// TwinCAT 3 PLC project PLC
// ProgramVersion: 3.1.4026.9
// CompilerDefines: {define InputField}{define ThirdOutputField}
// libraries:
//   Tc2_ControllerToolbox, * (Beckhoff Automation GmbH)
//   Tc2_ModbusRTU, * (Beckhoff Automation GmbH)
//   Tc2_ModbusSrv, * (Beckhoff Automation GmbH)
//   Tc2_Standard, * (Beckhoff Automation GmbH)
//   Tc2_System, * (Beckhoff Automation GmbH)
//   Tc2_Utilities, * (Beckhoff Automation GmbH)
//   Tc3_Module, * (Beckhoff Automation GmbH)
// project tree:
//   GVLs/ Config.TcGVL, GVL.TcGVL
//   / PlcTask.TcTTO
//   POUs/ErrorHandling/ eErrAckAccess.TcDUT, ErrorHandling.TcPOU, eSeverity.TcDUT, FB_AddErrorST.TcPOU, ST_ErrorStruct.TcDUT
//   POUs/ErrorHandling/New eventlogger %28TBD%29/ EventLogger.TcPOU (not stored), FB_Alarm.TcPOU (not stored), fb_EventAlarm.TcPOU (not stored)
//   POUs/FunctionBlocks/ fbDwordToReal.TcPOU, fbRealToDWord.TcPOU, fbRealToWord.TcPOU, fbWordToReal.TcPOU
//   POUs/ MAIN.TcPOU, POU.TcPOU
//   POUs/MonitoringControl/ FB_ControlManager.TcPOU
//   POUs/MonitoringControl/ProfinetController/enums/ e_controllerStatus.TcDUT
//   POUs/MonitoringControl/ProfinetController/ FB_PNController.TcPOU (excluded from build)
//   POUs/MonitoringControl/ProfinetController/Structs/future use/ ST_PNInput_DCBusExpansion.TcDUT, ST_PNInput_DCCharger.TcDUT, ST_PNInput_ParallelOperation.TcDUT, ST_PNOutput_DCCharger.TcDUT, ST_PNOutput_DCExpansion.TcDUT, ST_PNOutput_ParallelOperation.TcDUT
//   POUs/MonitoringControl/ProfinetController/Structs/ STParams.TcDUT, ST_PNController_Events.TcDUT, ST_PNController_Get.TcDUT, ST_PNController_Set.TcDUT, ST_PNInput_Battery.TcDUT, ST_PNInput_General.TcDUT, ST_PNInput_InputField.TcDUT, ST_PNInput_PeakShaveBox.TcDUT, ST_PNInput_Powerstack.TcDUT, ST_PNOutput_Battery.TcDUT, ST_PNOutput_General.TcDUT, ST_PNOutput_InputField.TcDUT, ST_PNOutput_OutputField.TcDUT, ST_PNOutput_PeakShaveBox.TcDUT, ST_PNOutput_PowerStack.TcDUT, ST_PNOutput_ZPT.TcDUT
//   POUs/Objects/BMS/eNums/ eBMS_Status.TcDUT, eHVDC_Powerstatus.TcDUT, ePOUState.TcDUT, ePowerControl.TcDUT, ePowerOnStatus.TcDUT, eSubValues.TcDUT
//   POUs/Objects/BMS/ FB_BMS.TcPOU, FB_BMS_IO.TcPOU
//   POUs/Objects/BMS/Structs/ st_BMS_Events.TcDUT, st_BMS_GetStatus.TcDUT, st_BMS_IO.TcDUT, st_BMS_Set.TcDUT, st_MBMU_BatterySummary.TcDUT, st_MBMU_Status.TcDUT, st_SBMU_BatterySummary.TcDUT, st_SBMU_Status.TcDUT
//   POUs/Objects/CoolingSystem/CoolingStack/eNums/ eHeatPumpMode.TcDUT, eHeatPumpState.TcDUT
//   POUs/Objects/CoolingSystem/CoolingStack/ FB_Heatpump.TcPOU, FB_HeatPumpSystem.TcPOU, FB_Heatpumpsystem_IO.TcPOU
//   POUs/Objects/CoolingSystem/CoolingStack/SFC/ FB_HeatpumpInit.TcPOU, FB_HeatpumpOperation.TcPOU
//   POUs/Objects/CoolingSystem/CoolingStack/Structs/ ST_HeatPumpSystemEvents.TcDUT, ST_HeatpumpSystemGet.TcDUT, ST_HeatpumpData.TcDUT, ST_HeatPumpEvents.TcDUT, ST_HeatPumpGet.TcDUT, st_OperatingPoint.TcDUT
//   POUs/Objects/CoolingSystem/ CoolingSystemParams.TcGVL, FB_CoolingSystem.TcPOU, FB_CoolingSystem_IO.TcPOU
//   POUs/Objects/CoolingSystem/SFC/Enums/ eConditioningRequirement.TcDUT, eConditioningStates.TcDUT
//   POUs/Objects/CoolingSystem/SFC/ FB_BatteryConditioningSFC.TcPOU, FB_DehumidifySFC.TcPOU, FB_EnclosureConditioningSFC.TcPOU, FB_PowerModeConditioningSFC.TcPOU
//   POUs/Objects/CoolingSystem/Structs/ ST_ConditioningRequirements.TcDUT, ST_CoolingSystemEvents.TcDUT, ST_CoolingSystemGet.TcDUT, ST_CoolingSystemInputs.TcDUT, ST_CoolingSystemOutputs.TcDUT, ST_CoolingSystem_Control.TcDUT, ST_SensorValues.TcDUT
//   POUs/Objects/ExternalControl/ FB_ExternalControl.TcPOU
//   POUs/Objects/InternalPowerSupply/eNums/ ePowerStatus.TcDUT, eSupplyState.TcDUT
//   POUs/Objects/InternalPowerSupply/ FB_InternalPowerSupply.TcPOU, FB_InternalPowerSupply_IO.TcPOU, IPSParams.TcGVL
//   POUs/Objects/InternalPowerSupply/Structs/ ST_InternalPowerStatus.TcDUT, ST_InternalPowerSupply_Events.TcDUT, ST_InternalPowerSupply_Get.TcDUT, ST_InternalPowersupply_set.TcDUT, ST_PowerDemand.TcDUT
//   POUs/Objects/InternalPowerSupply/UPS/eNums/ eUPSState.TcDUT
//   POUs/Objects/InternalPowerSupply/UPS/ FB_UPS.TcPOU
//   POUs/Objects/InternalPowerSupply/UPS/Structs/ ST_UPSData.TcDUT, ST_UPSEvents.TcDUT, ST_UPSGET.TcDUT
//   POUs/Objects/LedstripController/ eLedStripCommands.TcDUT, UpdateSFC.TcPOU
//   POUs/Objects/LedstripController/Structs/ stLedControl.TcDUT, stLedStatus.TcDUT, st_LedColor.TcDUT, ST_Ledstrip_IOvars.TcDUT, u_LedColor.TcDUT
//   POUs/Objects/PowerQualityMonitor/FB_Beckhoff_EL3443_0010/ FB_EL3443_0010.TcPOU, ST_EL3443_PhaseStatus.TcDUT, ST_EL3443_TotalStatus.TcDUT
//   POUs/Objects/PowerQualityMonitor/FB_Janitza_UMG801/ FB_Janitza.TcPOU, PowerMeterConfig.TcGVL, ST_Powerlockdata.TcDUT
//   POUs/Objects/PowerQualityMonitor/ FB_PowerQualityMonitoring.TcPOU
//   POUs/Objects/PowerQualityMonitor/_Enums/ eACRotationState.TcDUT, Phases.TcDUT
//   POUs/Objects/PowerQualityMonitor/_Structs/ ST_InputVoltageMeter.TcDUT, ST_PowerMonitor_BESS.TcDUT, ST_PowerMonitor_Events.TcDUT, ST_PowerMonitor_get.TcDUT, ST_PowerMonitor_InputField.TcDUT, ST_PowerMonitor_Internal.TcDUT, ST_PowerMonitor_OutputField.TcDUT
//   POUs/Objects/PowerStack/eNums/ eNetcontactorState.TcDUT, eStatus.TcDUT
//   POUs/Objects/PowerStack/ st_Powerstack_get.TcDUT
//   POUs/Objects/ProtectionSystems/FireDetection/eNums/ eFireAlarmStatus.TcDUT, eCOAlarmStatus.TcDUT
//   POUs/Objects/ProtectionSystems/FireDetection/ FB_FireDetection.TcPOU, FB_FireDetection_IO.TcPOU
//   POUs/Objects/ProtectionSystems/FireDetection/Structs/ ST_COInputData.TcDUT, ST_FireDetectionGet.TcDUT, ST_FireDetectionSet.TcDUT, ST_FireSystem_Events.TcDUT, ST_SmokeDetIO.TcDUT
//   POUs/Objects/RouterData/ FB_Teltonika.TcPOU
//   POUs/Objects/RouterData/Struct/ dwtoreal.TcDUT, eSMSStatus.TcDUT, st_Device.TcDUT, st_GPS.TcDUT, st_mobile.TcDUT, st_router_data.TcDUT, ST_Router_params.TcDUT, st_TeltonikaEvents.TcDUT
//   POUs/old/ old.TcPOU
//   POUs/ProfinetHandling/ InitSIEMENSInput.TcPOU, SetSiemensControlModes.TcPOU, SetSIEMENSOutput.TcPOU, SiemensControl.TcPOU
//   POUs/System/_Structs/ ST_SystemControl_FromSystem.TcDUT
//   POUs/System/_Structs/TempStructs/ eCOAlarmStatus_1.TcDUT, eSmokeDetectAlarmStatus.TcDUT, eWago750495_ACDataID.TcDUT, eWago750495_HarmonicsDataID.TcDUT, eWago750495_MeasureGroupID.TcDUT, eWago750495_StatDataID.TcDUT, ST_ACSwitchgear_Get.TcDUT, ST_CODetectors.TcDUT, ST_DCSwitchgear_Get.TcDUT, ST_Enclosure_get.TcDUT, ST_FireDetection_get.TcDUT, ST_FireDetection_get_1.TcDUT, ST_FireDetection_set.TcDUT, ST_FireSystem_Events_1.TcDUT, ST_FireSystem_Events_2.TcDUT, ST_InsulationMonitor_get.TcDUT, ST_NeutralTransformer_Get.TcDUT, ST_OvercurrentProtection_get.TcDUT, ST_PeakShaveBox_Get.TcDUT, ST_PLCstate_get.TcDUT, ST_ProtectionSystems_get.TcDUT, ST_ResidualCurrentMonitor_get.TcDUT, ST_Safety_get.TcDUT, ST_Safety_get_1.TcDUT, ST_SmokeDetectors.TcDUT, ST_SmokeDetIO_1.TcDUT, ST_Surgeprotection_get.TcDUT, ST_SystemControl_System.TcDUT, ST_System_Properties.TcDUT, ST_Wago750354_get.TcDUT, ST_Wago750495_Data.TcDUT, ST_Wago750495_ExtStatusWord.TcDUT, ST_Wago750495_Get.TcDUT, ST_Wago750495_Set.TcDUT, ST_Wago750495_StatusWord.TcDUT
// real-time tasks:
//   TASK PlcTask: cycle T#4ms, priority 1, ADS port 350
// I/O:
//   DEVICE Device 1 (EtherCAT), AmsNetId 5.131.105.63.2.1
//     Term 2 (EK1200) [EK1200-5000 EtherCAT Power supply (2A E-Bus)]
//       Term 2 (EL6070-0033) [EL6070-0033 1Ch. Licence key terminal, individual licences]
//       Term 25 (EL2574) [EL2574 4 Ch. Pixel LED Controller]
//         modules: SlotGroup 1 (Slot 1, 2), SlotGroup 1 (Slot 1, 2), SlotGroup 2 (Slot 3, 4), SlotGroup 2 (Slot 3, 4)
//       Term 3 (EL1809) [EL1809 16Ch. Dig. Input 24V, 3ms]
//       Term 4 (EL1809) [EL1809 16Ch. Dig. Input 24V, 3ms]
//       Term 6 (EL2809) [EL2809 16Ch. Dig. Output 24V, 0.5A]
//       Term 8 (EL2809) [EL2809 16Ch. Dig. Output 24V, 0.5A]
//       Term 9 (EL3054) [EL3054 4Ch. Ana. Input 4-20mA]
//       Term 10 (EL3054) [EL3054 4Ch. Ana. Input 4-20mA]
//       Term 11 (EL6021) [EL6021 Schnittstelle (RS422/485)]
//       Term 12 (EL3443-0010) [EL3443-0010 3Ch. Power Measuring 10A]
//       Term 13 (EL4002) [EL4002 2K. Ana. Ausgang 0-10V, 12bit]
//       Term 14 (EL1918) [EL1918, 8Ch. Safety Input 24V, TwinSAFE]
//         modules: Module 1 (FSOE), Module 2 (FSLOGIC)
//       Term 15 (EL2904) [EL2904, 4 Ch. Safety Output 24V, 0.5A, TwinSAFE]
//         modules: Module 1 (FSOES), Module 2 (DO)
//       Term 16 (EK1122) [EK1122 2 port EtherCAT junction]
//       Term 16 (EL9011) [EL9011 End Terminal]
//   DEVICE Device 4 (USB) (disabled)
//   DEVICE Device 5 (COM Port) (disabled)
//   DEVICE Device 6 (NOV-DP-RAM)
//   DEVICE Device 2 (Profinet Controller), AmsNetId 5.131.105.63.3.1
//     pn-coupler [Helmholz GmbH & Co. KG PN/PN Coupler X1 (left network), firmware V2, 700-158-3PN02, supports Conformance Class A,B 700-158-3PN02] (disabled)
//       modules: Term 3 (DAP Module), Term 4 (IN  32 Bytes), Term 5 (IN  32 Bytes), Term 7 (IN  32 Bytes), Term 8 (IN  32 Bytes), Term 9 (IN  32 Bytes), Term 10 (IN  64 Bytes), Term 11 (IN  64 Bytes), Term 16 (OUT  32 Bytes), Term 15 (OUT  64 Bytes), Term 14 (OUT  64 Bytes), Term 13 (OUT  64 Bytes), InOutPowerData (OUT 128 Bytes)
//     quint4-ups-24dc-24dc-40-pn [Phoenix Contact PROFINET IO - Uninterruptible Power Supply 2907079] (disabled)
//       modules: Term 1 (DAP Module), Term 2 (QUINT4-UPS 24DC/40)
//     pnpncouplerx1 [Helmholz GmbH & Co. KG PN/PN Coupler X1 (left network), firmware V2, 700-158-3PN02, supports Conformance Class A,B 700-158-3PN02] (disabled)
//       modules: Term 17 (DAP Module), Term 18 (PeakShaveBox)
//     pnmbcold [Helmholz GmbH & Co. KG PN/ModbusTCP Coupler V2, supports Conformance Class A,B 700-159-3MB02] (disabled)
//       modules: Term 6 (DAP Module), Term 19 (Write Holding Register), Term 20 (Read Holding Register)
//     pnpncouplerx1-20 [Helmholz GmbH & Co. KG PN/PN Coupler X1 (left network), firmware V2, 700-158-3PN02, supports Conformance Class A,B 700-158-3PN02] (disabled)
//       modules: Term 21 (DAP Module), Term 22 (General), Term 23 (Battery), Term 24 (OutputField), Term 25 (InputField)
//     pninternal [VDL energy systems PN/PN Coupler X1 (left network), firmware V2, 700-158-3PN02, supports Conformance Class A,B PNController] (disabled)
//       modules: Term 26 (DAP Module), Term 28 (General), Term 29 (Battery), Term 30 (OutputField), Term 31 (InputGeneratorField), Term 32 (PowerstackField), Term 33 (PeakShaveBoxField), Term 34 (NeutralTransformerField)
//     pnexternal [VDL energy systems PN/PN Coupler X2 (right network), firmware V2, 700-158-3PN02, supports Conformance Class A,B PNController] (disabled)
//       modules: Term 27 (DAP Module), Term 35 (General), Term 36 (Battery), Term 37 (OutputField), Term 38 (InputGeneratorField), Term 39 (PowerstackField), Term 40 (NeutralTransformerField)
//     pnmbc2 [Helmholz GmbH & Co. KG PN/ModbusTCP Coupler V2, supports Conformance Class A,B 700-159-3MB02] (disabled)
//       modules: Term 41 (DAP Module), General.SystemState, General.Status, General.Warnings, General.Errors, General.CS_Status, General.CS_Warnings, General.CS_Errors, General.IPS_Status, General.IPS_Warnings, General.IPS_Errors, General.HeartbeatOut, General.Control, General.HeartbeatIn
//     pnmbc [Helmholz GmbH & Co. KG PN/ModbusTCP Coupler V2, supports Conformance Class A,B 700-159-3MB02]
//       modules: Term 41 (DAP Module), General_out, General_in, BMS_out, BMS_in, OutputField_out, InputField_out, InputField_in, PowerStack_out, PowerStack_in, PSB_out, PSB_in, ZPT_out
// variable links:
//   PLC/PLC Instance <-> Device 1 (EtherCAT)/Term 2 (EK1200)/Term 25 (EL2574)
//     PlcTask Inputs/MAIN.LedStripSFC.st_Status/b_CMDReject <-> SlotGroup 1 (Slot 1, 2)/Status Channel %C/Status/Command Reject
//     PlcTask Inputs/MAIN.LedStripSFC.st_Status/b_Error <-> SlotGroup 1 (Slot 1, 2)/Status Channel %C/Status/Error
//     PlcTask Inputs/MAIN.LedStripSFC.st_Status/b_SendAck <-> SlotGroup 1 (Slot 1, 2)/Status Channel %C/Status/Send Acknowledge
//     PlcTask Inputs/MAIN.LedStripSFC.st_Status/b_Transmit <-> SlotGroup 1 (Slot 1, 2)/Status Channel %C/Status/Transmit
//     PlcTask Inputs/MAIN.LedStripSFC.st_Status/b_UpdateAck <-> SlotGroup 1 (Slot 1, 2)/Status Channel %C/Status/Update Acknowledge
//     PlcTask Inputs/MAIN.LedStripSFC.st_Status/b_Warning <-> SlotGroup 1 (Slot 1, 2)/Status Channel %C/Status/Warning
//     PlcTask Inputs/MAIN.LedStripSFC.st_Status/b_busy <-> SlotGroup 1 (Slot 1, 2)/Status Channel %C/Status/Busy
//     PlcTask Outputs/MAIN.LedStripSFC.st_Control/b_Execute <-> SlotGroup 1 (Slot 1, 2)/Control Channel %C/Control/Execute
//     PlcTask Outputs/MAIN.LedStripSFC.st_Control/b_Send <-> SlotGroup 1 (Slot 1, 2)/Control Channel %C/Control/Send
//     PlcTask Outputs/MAIN.LedStripSFC.st_Control/b_Update <-> SlotGroup 1 (Slot 1, 2)/Control Channel %C/Control/Update
//     PlcTask Outputs/MAIN.LedStripSFC.st_Control/by_Command <-> SlotGroup 1 (Slot 1, 2)/Control Channel %C/Control/Command
//     PlcTask Outputs/MAIN.LedStripSFC.st_Control/dw_Color <-> SlotGroup 1 (Slot 1, 2)/Control Channel %C/Control/Color
//     PlcTask Outputs/MAIN.LedStripSFC.st_Control/w_Index <-> SlotGroup 1 (Slot 1, 2)/Control Channel %C/Control/Index
//     PlcTask Outputs/MAIN.LedStripSFC.st_Control/w_Length <-> SlotGroup 1 (Slot 1, 2)/Control Channel %C/Control/Length
//     PlcTask Outputs/MAIN.LedStripSFC.st_Control/w_Parameter <-> SlotGroup 1 (Slot 1, 2)/Control Channel %C/Control/Parameter
//   PLC/PLC Instance <-> Device 2 (Profinet Controller)/pnmbc2
//     PlcTask Inputs/MAIN.MBTestin <-> API/General.HeartbeatIn/Subterm 78 (Read Holding Register)/Inputs/General.HeartbeatIn
//     PlcTask Outputs/MAIN.MBTestOut <-> API/General.HeartbeatOut/Subterm 76 (Write Holding Register)/Outputs/General.HeartbeatOut

CONFIGURATION PLC
    RESOURCE PLC ON TwinCAT3
        TASK PlcTask(INTERVAL := T#4ms, PRIORITY := 1);
        PROGRAM MAIN WITH PlcTask : MAIN;
    END_RESOURCE
END_CONFIGURATION

// ---- POUs/ErrorHandling/eErrAckAccess.TcDUT
{attribute 'qualified_only'}
{attribute 'strict'}
TYPE eErrAckAccess :
(
	General := 0,
	Operator := 1,
	VDL := 2
);
END_TYPE

// ---- POUs/ErrorHandling/eSeverity.TcDUT
{attribute 'qualified_only'}
{attribute 'to_string'}
TYPE eSeverity :
(
	EmergencyShutdown			:= 0, //ONLY CALL FROM SAFETY PROGRAM
	QuickShutdown				:= 1,			
	NormalShutdown				:= 2,
	Warning 					:= 3,
	Info						:= 4
);
END_TYPE

// ---- POUs/ErrorHandling/ST_ErrorStruct.TcDUT
TYPE ST_ErrorStruct :
STRUCT
	b_ErrorActive	:BOOL;
	s_Severity 		:STRING(20);
	s_ID			:STRING(4);
	s_Message		:STRING(100);
	s_DateError		:STRING(20);
	s_TimeError		:STRING(20);
	s_TimeCleared	:STRING(20);
END_STRUCT
END_TYPE

// ---- POUs/MonitoringControl/ProfinetController/enums/e_controllerStatus.TcDUT
{attribute 'qualified_only'}
{attribute 'strict'}
TYPE e_controllerStatus :
(
	None 	:= 	0,
	Init	:=	1,
	Ready	:=	2,
	Active	:=	3,
	Error	:=	4
);
END_TYPE

// ---- POUs/MonitoringControl/ProfinetController/Structs/future use/ST_PNInput_DCBusExpansion.TcDUT
TYPE ST_PNInput_DCBusExpansion :
STRUCT
	ControlBits	:	DWORD;
END_STRUCT
END_TYPE

// ---- POUs/MonitoringControl/ProfinetController/Structs/future use/ST_PNInput_DCCharger.TcDUT
TYPE ST_PNInput_DCCharger :
STRUCT
	Controlbits	:	DWORD;
	//b_enable?
	//b_resetCharger
	//b_StartCharging
	Powerlimit	:	DWORD;
END_STRUCT
END_TYPE

// ---- POUs/MonitoringControl/ProfinetController/Structs/future use/ST_PNInput_ParallelOperation.TcDUT
TYPE ST_PNInput_ParallelOperation :
STRUCT
	Controlbits			:	DWORD;
	//b_DetectSlaves	
	r_ActivePower		:	DWORD;
	r_reactivePower		:	DWORD;
END_STRUCT
END_TYPE

// ---- POUs/MonitoringControl/ProfinetController/Structs/future use/ST_PNOutput_DCCharger.TcDUT
TYPE ST_PNOutput_DCCharger :
STRUCT
	statusbits		:	DWORD;
	ChargerStatus	:	DWORD;
	ChargePower		:	DWORD;
END_STRUCT
END_TYPE

// ---- POUs/MonitoringControl/ProfinetController/Structs/future use/ST_PNOutput_DCExpansion.TcDUT
TYPE ST_PNOutput_DCExpansion :
STRUCT
	statusbits	: DWORD;
	Busvoltage	: DWORD;
	RatedPower	: DWORD;
	LoadPercentage	: DWORD;
	CurrentPower	: DWORD;
END_STRUCT
END_TYPE

// ---- POUs/MonitoringControl/ProfinetController/Structs/future use/ST_PNOutput_ParallelOperation.TcDUT
TYPE ST_PNOutput_ParallelOperation :
STRUCT
	statusbits		:	DWORD;
	ActivePower		:	DWORD;
	ReactivePower	:	DWORD;
END_STRUCT
END_TYPE

// ---- POUs/MonitoringControl/ProfinetController/Structs/STParams.TcDUT
TYPE STParams :
STRUCT
	t_HbIncrementInterval	:	TIME	:= 	T#500MS;
	t_HbCommLostTimeout		:	TIME	:=	T#1S;
END_STRUCT
END_TYPE

// ---- POUs/MonitoringControl/ProfinetController/Structs/ST_PNController_Events.TcDUT
TYPE ST_PNController_Events :
STRUCT
	b_HeartBeatLost				:	BOOL;
	b_DataConfigurationFault	:	BOOL;
	b_NetworkConfigurationFault	:	BOOL;
	b_DeviceFault				:	BOOL;
END_STRUCT
END_TYPE

// ---- POUs/MonitoringControl/ProfinetController/Structs/ST_PNController_Get.TcDUT
TYPE ST_PNController_Get :
STRUCT
	eControllerStatus	:	e_ControllerStatus;
	
	events				:	ST_PNController_Events;
END_STRUCT
END_TYPE

// ---- POUs/MonitoringControl/ProfinetController/Structs/ST_PNController_Set.TcDUT
TYPE ST_PNController_Set :
STRUCT

END_STRUCT
END_TYPE

// ---- POUs/MonitoringControl/ProfinetController/Structs/ST_PNInput_Battery.TcDUT
TYPE ST_PNInput_Battery :
STRUCT
	ui_SocMinLimit	:	UINT	:=	100;
	ui_SocMaxLimit	:	UINT	:=	0;
END_STRUCT
END_TYPE

// ---- POUs/MonitoringControl/ProfinetController/Structs/ST_PNInput_General.TcDUT
TYPE ST_PNInput_General :
STRUCT
	W_Control		:	WORD;
	ui_HeartBeat	:	UINT;
END_STRUCT
END_TYPE

// ---- POUs/MonitoringControl/ProfinetController/Structs/ST_PNInput_InputField.TcDUT
TYPE ST_PNInput_InputField :
STRUCT
	w_Control				:	WORD;
	ui_FeedInCurrentLimit	:	UINT;
	ui_FeedOutCurrentLimit	:	UINT;
	ui_IdleChargePower 		:	UINT;
	ui_SocTarget			:	UINT;
	ui_SOCStart				:	UINT;
	ui_SOCStop				:	UINT;
	ui_BatterOverloadStart	:	UINT;
	ui_BatteryOverloadStop	:	UINT;
END_STRUCT
END_TYPE

// ---- POUs/MonitoringControl/ProfinetController/Structs/ST_PNInput_PeakShaveBox.TcDUT
TYPE ST_PNInput_PeakShaveBox :
STRUCT
	w_ControlBits			:	WORD;
	ui_FeedInCurrentLimit	:	UINT;
	ui_SupplyCurrentLimit	:	UINT;
	UI_IdleChargePower		:	UINT;
	UI_SOCTarget			:	UINT;
END_STRUCT
END_TYPE

// ---- POUs/MonitoringControl/ProfinetController/Structs/ST_PNInput_Powerstack.TcDUT
TYPE ST_PNInput_Powerstack :
STRUCT
	w_ControlBits			:	WORD;
	w_GridMode				:	WORD;
	w_PowerMode				:	WORD;	
	ui_NominalVoltage		:	UINT;
	ui_NominalFrequency		:	UINT;	
	i_Pset					:	INT;
	i_Qset					:	INT;
	ui_PFset				:	UINT;
	ui_FrequencyDroop		:	UINT;
	ui_VoltageDroop			:	UINT;
	ui_Pmax					:	UINT;
	ui_Pmin					:	UINT;
	ui_QMax					:	UINT;
	ui_QMin					:	UINT;
	ui_ACCurrentLimit		:	UINT;
	ui_ApparentPowerLimit	:	UINT;
	ui_PowerRampRate		:	UINT;
END_STRUCT
END_TYPE

// ---- POUs/MonitoringControl/ProfinetController/Structs/ST_PNOutput_Battery.TcDUT
TYPE ST_PNOutput_Battery :
STRUCT
	w_Status						:	WORD;
	w_Warnings						:	WORD;
	w_Faults						:	WORD;

	ui_SOC							: UINT;
	ui_SOH							: UINT;
	ui_DClinkVoltage 				: UINT;
	i_DClinkCurrent 				: INT;
	ui_MaxAllowedDischargeCurrent 	: UINT;
	ui_MaxAllowedChargeCurrent 		: UINT;
	i_MinCellTemperature 			: INT;
	i_MaxCellTemperature			: INT;
	ui_RemainingChargeEnergy 		: UINT;
	ui_RemainingDischargeEnergy 	: UINT;
	ui_HistAccChargeEnergy_high		: UINT;
	ui_HistAccChargeEnergy_low		: UINT;
	ui_HistAccDischargeEnergy_high	: UINT;
	ui_HistAccDischargeEnergy_low	: UINT;
END_STRUCT
END_TYPE

// ---- POUs/MonitoringControl/ProfinetController/Structs/ST_PNOutput_General.TcDUT
TYPE ST_PNOutput_General :
STRUCT
	w_SystemState				:	WORD;
	w_SystemStatus				:	WORD;	
	w_SystemWarnings			:	WORD;
	w_SystemFaults				:	WORD;
	w_CoolingSystemStatus		:	WORD;
	w_CoolingSystemWarnings		:	WORD;
	w_CoolingSystemFaults		:	WORD;
	w_InternalSupplyStatus		:	WORD;
	w_InternalSupplyWarnings	:	WORD;
	w_InternalSupplyFaults		:	WORD;
	ui_HeartBeatOut				:	UINT;
END_STRUCT
END_TYPE

// ---- POUs/MonitoringControl/ProfinetController/Structs/ST_PNOutput_InputField.TcDUT
TYPE ST_PNOutput_InputField :
STRUCT
	w_Status					:	WORD;
	w_Warnings					:	WORD;
	w_Faults					:	WORD;
	
	i_ActivePower				:	INT;
	i_ReactivePower				:	INT;
	ui_Frequency				:	UINT;
	ui_VoltageL1N				:	UINT;
	ui_VoltageL2N				:	UINT;
	ui_VoltageL3N				:	UINT;
	ui_VoltageL1L2				:	UINT;
	ui_VoltageL2L3				:	UINT;
	ui_VoltageL3L1				:	UINT;
	i_CurrentL1					:	INT;
	i_CurrentL2					:	INT;
	i_CurrentL3					:	INT;
	i_CurrentN					:	INT;
	ui_TotalEnergySupplied_high :	UINT;
	ui_TotalEnergySupplied_low 	:	UINT;
	ui_TotalEnergyConsumed_high :	UINT;
	ui_TotalEnergyConsumed_low	:	UINT;
END_STRUCT
END_TYPE

// ---- POUs/MonitoringControl/ProfinetController/Structs/ST_PNOutput_OutputField.TcDUT
TYPE ST_PNOutput_OutputField :
STRUCT
	w_Status						:	WORD;
	w_Warnings						:	WORD;
	w_Faults						:	WORD;
	
	i_ActivePower				:	INT;
	i_ReactivePower				:	INT;
	ui_Frequency				:	UINT;
	ui_VoltageL1N				:	UINT;
	ui_VoltageL2N				:	UINT;
	ui_VoltageL3N				:	UINT;
	ui_VoltageL1L2				:	UINT;
	ui_VoltageL2L3				:	UINT;
	ui_VoltageL3L1				:	UINT;
	i_CurrentL1					:	INT;
	i_CurrentL2					:	INT;
	i_CurrentL3					:	INT;
	i_CurrentN					:	INT;
	ui_TotalEnergySupplied_high :	UINT;
	ui_TotalEnergySupplied_Low 	:	UINT;
	ui_TotalEnergyConsumed_high :	UINT;
	ui_TotalEnergyConsumed_low 	:	UINT;
END_STRUCT
END_TYPE

// ---- POUs/MonitoringControl/ProfinetController/Structs/ST_PNOutput_PeakShaveBox.TcDUT
TYPE ST_PNOutput_PeakShaveBox :
STRUCT
	w_Status					:	WORD;
	w_Warnings					:	WORD;
	w_Faults					:	WORD;
	
	i_ActivePower				:	INT;
	i_ReactivePower				:	INT;
	ui_Frequency				:	UINT;
	ui_VoltageL1N				:	UINT;
	ui_VoltageL2N				:	UINT;
	ui_VoltageL3N				:	UINT;
	ui_VoltageL1L2				:	UINT;
	ui_VoltageL2L3				:	UINT;
	ui_VoltageL3L1				:	UINT;
	i_CurrentL1					:	INT;
	i_CurrentL2					:	INT;
	i_CurrentL3					:	INT;
	i_CurrentN					:	INT;
END_STRUCT
END_TYPE

// ---- POUs/MonitoringControl/ProfinetController/Structs/ST_PNOutput_PowerStack.TcDUT
TYPE ST_PNOutput_PowerStack :
STRUCT
	w_Status					:	WORD;
	w_Warnings					:	WORD;
	w_Faults					:	WORD;
	w_PowerStackStatus			:	WORD;
	w_InverterMode				: 	WORD;
	w_Powermode					: 	WORD;
	
	i_ActivePower				: INT;
	i_ReactivePower				: INT;
	ui_D7_Voltage				: UINT;
	ui_D7_frequency				: UINT;
	i_ACCurrent					: INT;
	i_ActivePowerSetpoint		: INT;
	i_ReactivePowerSetpoint		: INT;
	ui_PFSetpoint				: UINT;
	ui_LoadPercentage			: UINT;
	ui_RatedCurrent				: UINT;
	ui_RatedPower				: UINT;
END_STRUCT
END_TYPE

// ---- POUs/MonitoringControl/ProfinetController/Structs/ST_PNOutput_ZPT.TcDUT
TYPE ST_PNOutput_ZPT :
STRUCT
	w_Status					:	WORD;
	w_Warnings					:	WORD;
	w_Faults					:	WORD;
	ui_RatedPower				:	UINT;
	ui_PowerLoad				:	UINT;
	i_TransformerTemperature	:	INT;
END_STRUCT
END_TYPE

// ---- POUs/Objects/BMS/eNums/eBMS_Status.TcDUT
{attribute 'qualified_only'}
{attribute 'strict'}
TYPE eBMS_Status :
(
	Init := 0,
	Normal := 1,
	FullCharge := 2,
	FullDischarge := 3,
	Warning := 4,
	Fault := 5,
	Off	:=	6
);
END_TYPE

// ---- POUs/Objects/BMS/eNums/eHVDC_Powerstatus.TcDUT
{attribute 'qualified_only'}
{attribute 'strict'}
TYPE eHVDC_Powerstatus :
(
	OFF := 0,
	Precharging := 1,
	ON	:= 2	
);
END_TYPE

// ---- POUs/Objects/BMS/eNums/ePOUState.TcDUT
{attribute 'qualified_only'}
{attribute 'strict'}
TYPE ePOUState :
(
	OFF := 0,
	PowerUp := 1,
	Init := 2,
	Normal	:=	3,
	EMSTOP	:=	4,
	Shutdown := 5
);
END_TYPE

// ---- POUs/Objects/BMS/eNums/ePowerControl.TcDUT
{attribute 'qualified_only'}
{attribute 'strict'}
TYPE ePowerControl :
(
	Init := 0,
	Stay := 1,
	PowerOn := 2,
	PowerOff := 3
)word;
END_TYPE

// ---- POUs/Objects/BMS/eNums/ePowerOnStatus.TcDUT
{attribute 'qualified_only'}
{attribute 'strict'}
TYPE ePowerOnStatus :
(
	Off := 0,
	On	:= 1,
	PowerOn_Fault := 2,
	PowerOff_Fault := 3
)UINT;
END_TYPE

// ---- POUs/Objects/BMS/eNums/eSubValues.TcDUT
{attribute 'qualified_only'}
{attribute 'strict'}
TYPE eSubValues :
(
	Minimum := 0,
	Average := 1,
	Maximum := 2
);
END_TYPE

// ---- POUs/Objects/BMS/Structs/st_BMS_Events.TcDUT
TYPE st_BMS_Events :
STRUCT
	//sunspec error list
	b_COMMUNICATION_ERROR			:	BOOL;
	b_OVER_TEMP_ALARM				:	BOOL;
	b_OVER_TEMP_WARNING				:	BOOL;
	b_UNDER_TEMP_ALARM				:	BOOL;
	b_UNDER_TEMP_WARNING			:	BOOL;
	b_OVER_CHARGE_CURRENT_ALARM		:	BOOL;
	b_OVER_CHARGE_CURRENT_WARNING	:	BOOL;
	b_OVER_DISCHARGE_CURRENT_ALARM	:	BOOL;
	b_OVER_DISCHARGE_CURRENT_WARNING:	BOOL;
	b_OVER_VOLT_ALARM				:	BOOL;
	b_OVER_VOLT_WARNING				:	BOOL;
	b_UNDER_VOLT_ALARM				:	BOOL;
	b_UNDER_VOLT_WARNING			:	BOOL;
	b_UNDER_SOC_MIN_ALARM			:	BOOL;
	b_UNDER_SOC_MIN_WARNING			:	BOOL;
	b_OVER_SOC_MAX_ALARM			:	BOOL;
	b_OVER_SOC_MAX_WARNING			:	BOOL;
	b_VOLTAGE_IMBALANCE_WARNING		:	BOOL;
	b_TEMPERATURE_IMBALANCE_ALARM	:	BOOL;
	b_TEMPERATURE_IMBALANCE_WARNING	:	BOOL;
	b_CONTACTOR_ERROR				:	BOOL;
	b_FAN_ERROR						:	BOOL;
	b_GROUND_FAULT					:	BOOL;
	b_OPEN_DOOR_ERROR				:	BOOL;
	b_CURRENT_IMBALANCE_WARNING		:	BOOL;
	b_OTHER_ALARM					:	BOOL;
	b_OTHER_WARNING					:	BOOL;
	b_CONFIGURATION_ALARM			:	BOOL;
	b_CONFIGURATION_WARNING			:	BOOL;

	(* old event list. Replaced by sunspec
	BMSWatchdogWarning				:	BOOL;
	BMSWatchdogError				:	BOOL;
	
	BMSWarningStatus				:	BOOL;
	BMSFaultStatus					:	BOOL;
	
	BMSPowerOnFault					:	BOOL;
	BMSPowerOffFault				:	BOOL;
	
	SOCLowWarning					: 	BOOL;
	OverVoltageWarning				:	BOOL;
	UnderVoltageWarning				:	BOOL;
	VoltageBalanceWarning			:	BOOL;
	
	OverTemperatureWarning			:	BOOL;
	UnderTemperatureWarning			:	BOOL;
	TemperatureDifferenceWarning	:	BOOL;
	
	OverCurrentWarning				:	BOOL;
	
	CommunicationWarning			:	BOOL;
	
	OverVoltageError				:	BOOL;
	UnderVoltageError				:	BOOL;
	OverTemperatureError			:	BOOL;
	UnderTemperatureError			:	BOOL;
	
	CSCError						:	BOOL;
	SBMUError						:	BOOL;
	MBMUError						:	BOOL;
	
	CommunicationError				:	BOOL;
	*)
END_STRUCT
END_TYPE

// ---- POUs/Objects/BMS/Structs/st_BMS_GetStatus.TcDUT
TYPE st_BMS_GetStatus :
STRUCT
	//Battery info
	BattInfo					:	st_MBMU_BatterySummary;
	
	//detailed info	
	MBMU_Status					:	st_MBMU_Status;
	SBMU						:	ARRAY[0..3] OF st_SBMU_Status;
	
	Events						:	st_BMS_Events;
END_STRUCT
END_TYPE

// ---- POUs/Objects/BMS/Structs/st_BMS_IO.TcDUT
TYPE st_BMS_IO :
STRUCT
	b_BMS_24V_Enable			:	BOOL;
	b_BMS_230V_Enable			:	BOOL;
END_STRUCT
END_TYPE

// ---- POUs/Objects/BMS/Structs/st_BMS_Set.TcDUT
TYPE st_BMS_Set :
STRUCT
	b_EnableBMS				:	BOOL;
	b_HVDC_Required			: 	BOOL;
END_STRUCT
END_TYPE

// ---- POUs/Objects/BMS/Structs/st_MBMU_BatterySummary.TcDUT
TYPE st_MBMU_BatterySummary :
STRUCT
		//general
	b_BMSHeartBeatOK				:	BOOL;
	ui_BMS_PowerOnStatus			:	ePowerOnStatus;
	ui_BMS_Status					:	eBMS_Status;		

	r_SystemVoltage					:	REAL;
	r_SystemCurrent					:	REAL;
	r_SOC							:	REAL;
	r_SOH							:	REAL;
	CellVoltage						:	ARRAY[0..2] OF REAL;
	CellTemperature					:	ARRAY[0..2] OF REAL;
	r_MaxChargeCurrentAllowed		:	REAL;
	r_MaxDischargeCurrentAllowed	:	REAL;
	r_MaxChargePowerAllowed			:	REAL;
	r_MaxDischargePowerAllowed		:	REAL;
	r_MaxSystemVoltageAllowed		:	REAL;
	r_MinSystemVoltageAllowed		:	REAL;
	
	r_SystemPower					:	REAL;
	r_ChargeSOE						:	REAL;
	r_DischargeSOE					:	REAL;
	
	r_RemainingChargeEnergy			:	REAL;
	r_RemainingDischargeEnergy		:	REAL;
	
	r_HistAccChargeEnergy			:	REAL;
	r_HistAccDischargeEnergy		:	REAL;
END_STRUCT	
END_TYPE

// ---- POUs/Objects/BMS/Structs/st_MBMU_Status.TcDUT
TYPE st_MBMU_Status :
STRUCT
	GeneralSBMUStatus			:	ARRAY [0..15] OF WORD;
	MBMUStatus					:	ARRAY [0..15] OF WORD;

	s_MBMU_SWVer				:	STRING(16);
	s_MBMU_HWVer				:	STRING(16);
	
	s_ETH_SWVer					:	STRING(32);
	r_ETH_HWVer					:	STRING(32);	
	
	by_NumberOfSubSystems		:	BYTE;
	DateTime					:	ARRAY[0..5] OF WORD;
	b_InsulationSwitchOpen		:	BOOL;
	
	BatteryStatus				:	st_MBMU_BatterySummary;
END_STRUCT
END_TYPE

// ---- POUs/Objects/BMS/Structs/st_SBMU_BatterySummary.TcDUT
TYPE st_SBMU_BatterySummary :
STRUCT
	r_SystemVoltage			:	REAL;
	r_SystemCurrent			:	REAL;
	r_SOC					:	REAL;
	r_SOH					:	REAL;
	CellVoltage				:	ARRAY[0..2] OF REAL;
	CellTemperature			:	ARRAY[0..2] OF REAL;
	r_MaxChargeCurrentAllowed		:	REAL;
	r_MaxDischargeCurrentAllowed	:	REAL;
	r_HistAccChargeEnergy			:	REAL;
	r_HistAccDischargeEnergy		:	REAL;
	
	//Gaan we hier uberhaupt iets mee doen?
	w_MaxVoltageCellLocation 	: 	WORD;//ARRAY[0..1] OF BYTE;
	w_MinVoltageCellLocation 	:	 WORD;//ARRAY[0..1] OF BYTE;
	w_MaxTempCellLocation 		: 	WORD;//ARRAY[0..1] OF BYTE;
	w_MinTempCellLocation 		: 	WORD;//ARRAY[0..1] OF BYTE;
	r_SumOfCellVoltages			:	REAL;
END_STRUCT
END_TYPE

// ---- POUs/Objects/BMS/Structs/st_SBMU_Status.TcDUT
TYPE st_SBMU_Status :
STRUCT
	w_SystemWarning			:	WORD;
	SystemAlarm				:	ARRAY [0..2] OF WORD;
	
	b_PrechargeRelayClosed	:	BOOL;
	b_MainPosRelayClosed	:	BOOL;
	b_MainNegRelayClosed	:	BOOL;
	b_ControlBoxFanOn		:	BOOL;
	b_BalanceStatus			:	BOOL;
	b_DoorState				:	BOOL;	
	
	s_SBMU_SWVer			:	STRING(16);
	s_SBMU_HWVer			:	STRING(16);
	s_CSC_SWVer				:	STRING(16);
	s_CSC_HWVer				:	STRING(16);
	
	BatteryStatus			:	st_SBMU_BatterySummary;
END_STRUCT
END_TYPE

// ---- POUs/Objects/CoolingSystem/CoolingStack/eNums/eHeatPumpMode.TcDUT
{attribute 'qualified_only'}
{attribute 'strict'}
TYPE eHeatPumpMode :
(
	Standby := 0,
	Cooling := 1,
	Heating := 2
)UINT := Standby;
END_TYPE

// ---- POUs/Objects/CoolingSystem/CoolingStack/eNums/eHeatPumpState.TcDUT
{attribute 'qualified_only'}
{attribute 'strict'}
TYPE eHeatPumpState :
(
	OFF := 0,
	Initializing := 1,
	Standby := 2,
	Active_Cooling := 3,
	Active_Heating := 4,
	ERROR := 5
)UINT := OFF;
END_TYPE

// ---- POUs/Objects/CoolingSystem/CoolingStack/Structs/ST_HeatPumpSystemEvents.TcDUT
TYPE ST_HeatPumpSystemEvents :
STRUCT

END_STRUCT
END_TYPE

// ---- POUs/Objects/CoolingSystem/CoolingStack/Structs/ST_HeatpumpSystemGet.TcDUT
TYPE ST_HeatpumpSystemGet :
STRUCT
	HeatPumpStatus 			: 	eHeatPumpState;
	PrimaryHeatpumpGet		:	REFERENCE TO ST_HeatpumpGet;
	SecondaryHeatpumpGet 	:	REFERENCE TO ST_HeatpumpGet;
	//Heatpumps		:	REFERENCE TO ARRAY[1..2] OF ST_HeatPumpGet;
END_STRUCT
END_TYPE

// ---- POUs/Objects/CoolingSystem/CoolingStack/Structs/ST_HeatpumpData.TcDUT
TYPE ST_HeatpumpData :
STRUCT
	i_FW_Version		:	INT;		//1
	i_FW_release		:	INT;		//2
	w_FW_Subrelease		:	WORD;		//3
	w_FW_creationDate	:	WORD;		//4
	
	w_Serialnumber		:	ARRAY[0..17] OF WORD;	//80-97
	
	i_OperatingHours	:	INT;		//305-317?
	
	r_InletWaterTemp	:	REAL;		//400
	r_OutletWaterTemp	:	REAL;		//401
	r_HighPressure		:	REAL;		//406
	r_LowPressure		:	REAL;		//414
	r_CompInputTemp		:	REAL;		//422
	r_OutdoorTemp		:	REAL;		//428
	r_CompOutputTemp	:	REAL;		//433-435
	ui_WaterFlowRate	:	UINT;		//444
	
	w_ErrorList			:	ARRAY[1..7] OF WORD;	//950-956	
	
	r_FanSpeedPCT		:	REAL;		//7000
	r_PumpSpeedPCT		:	REAL;		//7001
	
	r_SetpointHeating	:	REAL;		//7204
	r_SetpointCooling	:	REAL;		//7203
	b_DefrostingActive	:	BOOL;		//7214.14
END_STRUCT
END_TYPE

// ---- POUs/Objects/CoolingSystem/CoolingStack/Structs/ST_HeatPumpEvents.TcDUT
TYPE ST_HeatPumpEvents :
STRUCT
	b_CommError			: BOOL;
	b_ProbeError		: BOOL;
	b_PressureError		: BOOL;
	b_CompressorError	: BOOL;
	b_ValveError		: BOOL;
	b_FanError			: BOOL;
	b_PumpError			: BOOL;
	b_WaterTempError	: BOOL;
	b_IOError			: BOOL;
	
	b_CommWarning		:	BOOL;
END_STRUCT
END_TYPE

// ---- POUs/Objects/CoolingSystem/CoolingStack/Structs/ST_HeatPumpGet.TcDUT
TYPE ST_HeatPumpGet :
STRUCT
	HeatPumpState 	: 	eHeatPumpState;
	Setpoint		:	REAL;
	Events			: 	ST_HeatPumpEvents;
	
	HeatpumpData	:	ST_HeatpumpData;
END_STRUCT
END_TYPE

// ---- POUs/Objects/CoolingSystem/CoolingStack/Structs/st_OperatingPoint.TcDUT
TYPE st_OperatingPoint :
STRUCT
	OperatingMode	:	eHeatpumpMode;
	Setpoint		:	REAL;
END_STRUCT
END_TYPE

// ---- POUs/Objects/CoolingSystem/SFC/Enums/eConditioningRequirement.TcDUT
{attribute 'qualified_only'}
{attribute 'strict'}
TYPE eConditioningRequirement :
(
	None := 0,
	Cooling := -1,
	Heating := +1
) int := None;
END_TYPE

// ---- POUs/Objects/CoolingSystem/SFC/Enums/eConditioningStates.TcDUT
{attribute 'qualified_only'}
{attribute 'strict'}
TYPE eConditioningStates :
(
	OFF 						:= 	0,
	EnclosureConditioning 		:= 	1,
	InverterZPTStartup 			:= 	2,
	BatteryConditioning 		:= 	3,
	DeHum 						:= 	4,
	InverterPowerMode 			:= 	5,
	EMSTOP						:=	6
)uint := OFF;
END_TYPE

// ---- POUs/Objects/CoolingSystem/Structs/ST_ConditioningRequirements.TcDUT
TYPE ST_ConditioningRequirements :
STRUCT
	by_PSCoolingPowerMode	:	BYTE;
	by_SetCooling			:	BYTE;
	Enclosure				:	eConditioningRequirement := 0;
	Battery					:	eConditioningRequirement := 0;
	Dehum					:	BOOL;
END_STRUCT
END_TYPE

// ---- POUs/Objects/CoolingSystem/Structs/ST_CoolingSystemEvents.TcDUT
TYPE ST_CoolingSystemEvents :
STRUCT
	b_SystemOvertemperatureWarning	:	BOOL;
	b_SystemUnderTemperatureWarning :	BOOL;
	
	//faults
	b_CoolingSystemFuseFailure		: 	BOOL;	
	
	b_InverterLoopValveStuck		: 	BOOL;
	b_BattLoopValveStuck			: 	BOOL;
	b_FancoilLoopValveStuck			: 	BOOL;
	
	//System pressure dropped below idle minimum pressure. suspect coolant loss.
	b_CoolingLoopIdlePressureWarning 	: 	BOOL := FALSE;	
	b_CoolingLoopIdlePressureError 		: 	BOOL := FALSE;	
	
	//Systempressure too low during conditioning, possible pump failure or coolant loss.
	b_InverterCoolingLoopError 		: 	BOOL := FALSE;

	b_HeatpumpWarning				:	BOOL;
	b_HeatPumpError					: 	BOOL;
END_STRUCT
END_TYPE

// ---- POUs/Objects/CoolingSystem/Structs/ST_CoolingSystemGet.TcDUT
TYPE ST_CoolingSystemGet :
STRUCT
	CoolingSystemMode		:	eConditioningStates;
	HeatPumpStatus			: 	eHeatPumpState;
	CoolantTemperature		:	REAL;
	CoolantPressure			:	REAL;
	EnclosureDewpoint		:	REAL;
		
	
	HeatPumpSystemGet 		: REFERENCE TO ST_HeatpumpSystemGet;	
	Events					: ST_CoolingSystemEvents;
END_STRUCT
END_TYPE

// ---- POUs/Objects/CoolingSystem/Structs/ST_CoolingSystemInputs.TcDUT
TYPE ST_CoolingSystemInputs :
STRUCT
	BattLoopValveFB					:	BOOL;
	InvLoopValveFB					:	BOOL;
	FancoilLoopValveFB				:	BOOL;
	
	CoolingLoopPressureSensor 		:	INT;
	CoolingLoopTemperatureSensor 	:	INT;
	
	CoolingSystem400VFuseFB			:	BOOL;
	
END_STRUCT
END_TYPE

// ---- POUs/Objects/CoolingSystem/Structs/ST_CoolingSystemOutputs.TcDUT
TYPE ST_CoolingSystemOutputs :
STRUCT
	DCFanEnable						:	BOOL;
	
	BattLoopValveClose				:	BOOL;
	InvLoopValveClose				:	BOOL;
	FancoilLoopValveClose			:	BOOL;
		
	DCPumpEnable					: 	BOOL;
	ACPumpEnable					: 	BOOL;
END_STRUCT
END_TYPE

// ---- POUs/Objects/CoolingSystem/Structs/ST_CoolingSystem_Control.TcDUT
TYPE ST_CoolingSystem_Control :
STRUCT
	//system outputs
	b_CloseBatteryLoopValve		:	BOOL;
	b_CloseInverterLoopValve	:	BOOL;
	b_CloseFancoilLoopValve 	:	BOOL;
	
	b_BatteryLoopEnabled		:	BOOL;
	b_InverterLoopEnabled		:	BOOL;
	b_FancoilLoopEnabled		:	BOOL;
	
	b_DCFancoilEnable			: 	BOOL;
	b_DCPumpEnable 				: 	BOOL;
	b_ACPumpEnable				: 	BOOL;
	
	//System inputs
	r_EnclosureHumidity			:	REAL;
	r_EnclosureTemperature		:	REAL;
	r_CoolantTemperature		:	REAL;
	
	r_CoolantPressure			:	REAL;
	r_CoolantIdlePressure		:	REAL;
	
	r_CurrentEnclosureDewPoint	: 	REAL;
	
	//Inputs via main sequence
	//From BMS
	r_BMSBatteryTemperature		:	REAL;
	R_BMSMaxBatteryTemperature	: 	REAL;
	
	//From PowerModule
	r_InverterTemperature		:	REAL;
	r_FilterTemperature			:	REAL;
	r_OutputPowerLevel			:	REAL;
	b_InverterRunning			: 	BOOL;
	
	//HeatpumpData
	b_HeatPumpPowerEnable		:	BOOL;
	r_HeatPumpSetpoint			:	REAL;
	e_HeatpumpMode				:	eHeatPumpMode;
	HeatPumpStatus				:	eHeatPumpState;
	
	//From Internal power supply
	b_24V_Available				:	BOOL; 
	b_400v_Available			:	BOOL;
END_STRUCT
END_TYPE

// ---- POUs/Objects/CoolingSystem/Structs/ST_SensorValues.TcDUT
TYPE ST_SensorValues :
STRUCT

END_STRUCT
END_TYPE

// ---- POUs/Objects/InternalPowerSupply/eNums/ePowerStatus.TcDUT
{attribute 'qualified_only'}
{attribute 'strict'}
(*
TYPE ePowerStatus :
(
	Off := 	0,
	On	:=	1,
	Fault	:=	2
);
*)

// ---- POUs/Objects/InternalPowerSupply/eNums/eSupplyState.TcDUT
{attribute 'qualified_only'}
{attribute 'strict'}
TYPE eSupplyState :
(
	enum_member := 0
);
END_TYPE

// ---- POUs/Objects/InternalPowerSupply/Structs/ST_InternalPowerStatus.TcDUT
TYPE ST_InternalPowerStatus :
STRUCT
	b_Status_24VDC		:	BOOL;
	b_Status_HVDC		:	BOOL;
	b_Status_400VAC		:	BOOL;
END_STRUCT
END_TYPE

// ---- POUs/Objects/InternalPowerSupply/Structs/ST_InternalPowerSupply_Events.TcDUT
TYPE ST_InternalPowerSupply_Events :
STRUCT
	b_DCPSUFault				: 	BOOL; //fuse blown or psu_ok signal lost
	b_ACPSUFault				: 	BOOL;
	b_GridInputFuseTripped		:	BOOL;
	b_CEEInputFuseTripped		:	BOOL;
	b_HVDCShutdownTimeExceeded	:	BOOL;
END_STRUCT
END_TYPE

// ---- POUs/Objects/InternalPowerSupply/Structs/ST_InternalPowerSupply_Get.TcDUT
TYPE ST_InternalPowerSupply_Get :
STRUCT
	b_24VdcAvailable	:	BOOL;
	b_HVDCAvailable		:	BOOL;
	b_400VACAvailable	:	BOOL;
	
	UPS				:	ST_UPSGet;	
	
	Events			:	st_InternalPowerSupply_Events;
END_STRUCT
END_TYPE

// ---- POUs/Objects/InternalPowerSupply/Structs/ST_InternalPowersupply_set.TcDUT
TYPE ST_InternalPowersupply_set :
STRUCT
	CoolingSystemPowerDemand	:	st_PowerDemand;
	PowerStackPowerDemand		:	st_PowerDemand;	
	UPSPowerDemand				:	st_PowerDemand;
	InternalPowerDemand			:	st_PowerDemand;
	
	b_GeneralPowerEnable			: 	BOOL 	:= FALSE;	//?
	
	b_InternalBusbarACAvailable		:	BOOL	:=	FALSE;
	
	b_ShutdownUPS		:	BOOL;
END_STRUCT
END_TYPE

// ---- POUs/Objects/InternalPowerSupply/Structs/ST_PowerDemand.TcDUT
TYPE ST_PowerDemand :
STRUCT
	b_Demand_24V	:	BOOL;
	b_Demand_400V	:	BOOL;
	b_Demand_HVDC	:	BOOL;
END_STRUCT
END_TYPE

// ---- POUs/Objects/InternalPowerSupply/UPS/eNums/eUPSState.TcDUT
{attribute 'qualified_only'}
{attribute 'strict'}
TYPE eUPSState :
(
	Inoperative 	:= 0,
	Input_Active	:= 1,
	On_Battery		:= 2
);
END_TYPE

// ---- POUs/Objects/InternalPowerSupply/UPS/Structs/ST_UPSData.TcDUT
TYPE ST_UPSData :
STRUCT
	udi_StatusFunctions 		: 	UDINT;
	udi_StatusInterface 		: 	UDINT;
	ui_InputVoltage				:	UINT;
	ui_InputCurrent				:	UINT;
	ui_OutputVoltage			:	UINT;
	ui_OutputCurrent			:	UINT;
	ui_BatteryVoltage			: 	UINT;
	ui_BatteryChargingCurrent 	: 	UINT;
	ui_BatteryTemperature 		: 	UINT;
	ui_DeviceTemperature		: 	UINT;
	udi_SOC 					:	UDINT;
	ui_TuPCShutdown				:	UINT;
	ui_SOH						:	UINT;
	ui_PHStatus					:	UINT;
	ui_DEVOPTIME				:	UINT;
	ui_DEVUSEROPTIME			:	UINT;
	ui_DEVSTARTS				:	UINT;
END_STRUCT
END_TYPE

// ---- POUs/Objects/InternalPowerSupply/UPS/Structs/ST_UPSEvents.TcDUT
TYPE ST_UPSEvents :
STRUCT
	b_BatteryLowNotice		:	BOOL;	//initialize DC conditioning
	b_BatteryLowWarning		:	BOOL;	//Battery charging failed, consider shutdown
	b_BatteryLowError		:	BOOL;	//Battery level critical, System should shutdown
	b_NoBatteryError		:	BOOL;	//no Battery voltage detected?
	b_InputVoltageError		:	BOOL;	//ipsstate says 24v is available, but no input is seen.
END_STRUCT
END_TYPE

// ---- POUs/Objects/InternalPowerSupply/UPS/Structs/ST_UPSGET.TcDUT
TYPE ST_UPSGET :
STRUCT
	r_InputVoltage		:	REAL;
	r_OutputVoltage		:	REAL;
	r_BatteryVoltage	:	REAL;
	ui_SOC				:	UINT;
	
	b_ChargerActive		:	BOOL;
	b_SystemOnBattery	:	BOOL;
	
	UPSPowerDemand	:  	ST_PowerDemand;
	
	Events			:	ST_UPSEvents;
END_STRUCT
END_TYPE

// ---- POUs/Objects/LedstripController/eLedStripCommands.TcDUT
{attribute 'qualified_only'}
{attribute 'strict'}
TYPE eLedStripCommands :
(
	NOP 		:= 	0,
	Fill		:=	1,
	ClearAll	:=	2,
	CopyPixels	:=	3,
	MOVEPixels	:=	4,
	ROLPixels	:=	5,
	RORPixels	:=	6,
	ReverseOrder	:=	7,
	GradientFirstColor	:=	8,
	GradientLastColor	:=	9	
) BYTE;
END_TYPE

// ---- POUs/Objects/LedstripController/Structs/stLedControl.TcDUT
TYPE stLedControl :
STRUCT
	b_Execute	:	BOOL;
	b_Send		:	BOOL;
	b_Update	:	BOOL;
	by_Command	:	BYTE;
	w_Index		:	WORD;
	w_Length	:	WORD;
	w_Parameter	:	WORD;
	dw_Color	:	DWORD;
END_STRUCT
END_TYPE

// ---- POUs/Objects/LedstripController/Structs/stLedStatus.TcDUT
TYPE stLedStatus :
STRUCT
	b_busy		:	BOOL;
	b_Transmit	:	BOOL;
	b_SendAck	:	BOOL;
	b_UpdateAck	:	BOOL;
	b_CMDReject	:	BOOL;
	b_Warning	:	BOOL;
	b_Error		:	BOOL;
END_STRUCT
END_TYPE

// ---- POUs/Objects/LedstripController/Structs/st_LedColor.TcDUT
TYPE st_LedColor :
STRUCT
	by_Red		:	BYTE;
	by_Green	:	BYTE;
	by_Blue		:	BYTE;
	by_White	:	BYTE;
END_STRUCT
END_TYPE

// ---- POUs/Objects/LedstripController/Structs/ST_Ledstrip_IOvars.TcDUT
TYPE ST_Ledstrip_IOvars :
STRUCT
	r_Soc						: REAL;
	b_Error						: BOOL;
	b_warning					: BOOL;
	b_attention					: BOOL;
	b_normal					: BOOL;
	r_DCCurrent					: REAL;
END_STRUCT
END_TYPE

// ---- POUs/Objects/LedstripController/Structs/u_LedColor.TcDUT
TYPE u_LedColor :
UNION
	dw_LedColor	:	DWORD;
	st_LedColor	:	st_LedColor;
END_UNION
END_TYPE

// ---- POUs/Objects/PowerQualityMonitor/FB_Beckhoff_EL3443_0010/ST_EL3443_PhaseStatus.TcDUT
TYPE ST_EL3443_PhaseStatus :
STRUCT
	bit_voltageSign				: BIT;
	bit_Overvoltage				: BIT;
	bit_Overcurrent           	: BIT;
	bit_InaccurateVoltage     	: BIT;
	bit_InaccurateCurrent     	: BIT;
	bit_VoltageGuardWarning   	: BIT;
	bit_VoltageGuardError     	: BIT;
	bit_CurrentGuardWarning   	: BIT;
	bit_CurrentGuardError     	: BIT;
	bit_TxPDOToggle           	: BIT;
END_STRUCT
END_TYPE

// ---- POUs/Objects/PowerQualityMonitor/FB_Beckhoff_EL3443_0010/ST_EL3443_TotalStatus.TcDUT
TYPE ST_EL3443_TotalStatus :
STRUCT
	bit_SystemState						: BIT;
	bit_GridDirection					: BIT;
	bit_FrequencyGuardWarning			: BIT;
	bit_FrequencyGuardError             : BIT;
	bit_NeutralCurrentGuardWarning      : BIT;
	bit_NeutralCurrentGuardError        : BIT;
	bit_ActivePowerGuardWarning         : BIT;
	bit_ActivePowerGuardError           : BIT;
	bit_ApparentPowerGuardWarning       : BIT;
	bit_ApparentPowerGuardError         : BIT;
	bit_PowerQualityGuardWarning        : BIT;
	bit_PowerQualityGuardError          : BIT;
	bit_TxPDOState                      : BIT;
	bit_TxPDOToggle                     : BIT;
	r_PowerQualityFactor				: REAL;
END_STRUCT
END_TYPE

// ---- POUs/Objects/PowerQualityMonitor/FB_Janitza_UMG801/ST_Powerlockdata.TcDUT
TYPE ST_Powerlockdata :
STRUCT
	//Power
	r_ApparentPhasePower	: 	ARRAY[0..3] OF REAL;
	r_ReactivePhasePower	: 	ARRAY[0..3] OF REAL;
	r_ActivePhasePower		: 	ARRAY[0..3] OF REAL;	

	//Power
	r_ApparentPower				: 	REAL := 0;
	r_ReactivePower				:	REAL := 0;
	r_ActivePower				:	REAL := 0; 	

	//Energy Consumed
	r_EnergyConsumed			:	REAL := 0;
	
	//Energy Delivered
	r_EnergySupplied			:	REAL := 0;
	
	//THD
	ar_THD						:	ARRAY[0..3] OF REAL := [0, 0, 0, 0];	

	ar_PowerFactor				:	ARRAY[0..3] OF REAL := [0, 0, 0, 0];
END_STRUCT
END_TYPE

// ---- POUs/Objects/PowerQualityMonitor/_Enums/eACRotationState.TcDUT
{attribute 'qualified_only'}
{attribute 'strict'}
TYPE eACRotationState :
(
	Left := -1,
	None := 0,
	Right := 1
);
END_TYPE

// ---- POUs/Objects/PowerQualityMonitor/_Enums/Phases.TcDUT
{attribute 'qualified_only'}
{attribute 'strict'}
TYPE Phases :
(
	AVG := 0,
	L1	:=	1,
	L2	:=	3,
	L3	:=	2,
	N	:=	4
);
END_TYPE

// ---- POUs/Objects/PowerQualityMonitor/_Structs/ST_InputVoltageMeter.TcDUT
TYPE ST_InputVoltageMeter :
STRUCT
	GenPhaseVoltage : ARRAY[1..3] OF REAL;
	GenLineVoltage : ARRAY[1..3] OF REAL;
	GenFrequency : REAL;
	GenFieldDirection: BOOL;
	EL3443Status	:	UINT;
END_STRUCT
END_TYPE

// ---- POUs/Objects/PowerQualityMonitor/_Structs/ST_PowerMonitor_BESS.TcDUT
TYPE ST_PowerMonitor_BESS :
STRUCT
	r_Current					:	ARRAY[0..4] OF REAL;
	
	//Power
	r_ApparentPower		: 	REAL;
	r_ReactivePower		: 	REAL;
	r_ActivePower		: 	REAL;
	
	//Power
	r_ApparentPhasePower	: 	ARRAY[0..3] OF REAL;
	r_ReactivePhasePower	: 	ARRAY[0..3] OF REAL;
	r_ActivePhasePower		: 	ARRAY[0..3] OF REAL;
	
	//Energy Consumed
	r_EnergyConsumed		:	REAL;
	
	//Energy Delivered
	r_EnergySupplied		:	REAL;
	
	r_THD						:	ARRAY[0..3] OF REAL;
	r_PowerFactor 				:	ARRAY[0..3] OF REAL;
	r_Frequency					: 	REAL;

	//--//Overcurrent quicklog
	b_OvercurrentDetected		:	BOOL; //general Flag
	w_OvercurrentPhases			:	WORD; // first 4 bits (OUT1: L1/L2/L3/N)
	ui_OvercurrentCount			: 	UINT;
	t_LastOverCurrentTimeStap	:	TIME;
	r_LastOvercurrentDuration	:	REAL;
	t_MaxOvercurrentTimestamp	:	TIME;
END_STRUCT
END_TYPE

// ---- POUs/Objects/PowerQualityMonitor/_Structs/ST_PowerMonitor_Events.TcDUT
TYPE ST_PowerMonitor_Events :
STRUCT
	b_MBCommWarning 		: BOOL;
	b_MBCommError 			: BOOL;
	b_MBTimeoutWarning 		: BOOL;
	b_EL3443Warning			: BOOL;
	b_EL3443Error		: BOOL;
END_STRUCT
END_TYPE

// ---- POUs/Objects/PowerQualityMonitor/_Structs/ST_PowerMonitor_get.TcDUT
TYPE ST_PowerMonitor_get :
STRUCT
	PQMeterReady	: 	BOOL;
	InputField		:	ST_PowerMonitor_InputField;	
	OutputField		:	ST_PowerMonitor_OutputField;
	InternalSupply	:	ST_PowerMonitor_Internal;
	
	//Inverter power/energy input & output
	BESS			:	ST_PowerMonitor_BESS;

	
	events			:	ST_PowerMonitor_Events;
END_STRUCT
END_TYPE

// ---- POUs/Objects/PowerQualityMonitor/_Structs/ST_PowerMonitor_InputField.TcDUT
TYPE ST_PowerMonitor_InputField :
STRUCT
	e_ACrotationStatus	:	eACRotationState;
	r_Frequency			: 	REAL;

	r_PhaseVoltage		: 	ARRAY[0..3] OF REAL;
	r_LineVoltage		:	ARRAY[0..3] OF REAL;
	
	//Power
	r_ApparentPower		: 	REAL;
	r_ReactivePower		: 	REAL;
	r_ActivePower		: 	REAL;
	
	//Power
	r_ApparentPhasePower	: 	ARRAY[0..3] OF REAL;
	r_ReactivePhasePower	: 	ARRAY[0..3] OF REAL;
	r_ActivePhasePower		: 	ARRAY[0..3] OF REAL;

	//Energy Consumed
	r_EnergyConsumed		:	REAL;
	
	//Energy Delivered
	r_EnergySupplied		:	REAL;
	
	//currents
	r_Current					:	ARRAY[0..4] OF REAL;
	
	//THD
	r_THD						:	ARRAY[0..3] OF REAL;
		
	r_PowerFactor				:	ARRAY[0..3] OF REAL;
	
	//PowerLock Currents, 2 fields of 4 measurements
	ar_PowerlockCurrents		: 	ARRAY [1..2] OF ARRAY[1..4] OF REAL;
END_STRUCT
END_TYPE

// ---- POUs/Objects/PowerQualityMonitor/_Structs/ST_PowerMonitor_Internal.TcDUT
TYPE ST_PowerMonitor_Internal :
STRUCT
	e_ACrotationStatus	:	eACRotationState;
	r_Frequency			: 	REAL;
	
	r_PhaseVoltage		: 	ARRAY[0..3] OF REAL;
	r_LineVoltage		:	ARRAY[0..3] OF REAL;
	
	//Power
	r_ApparentPower		: 	REAL;
	r_ReactivePower		: 	REAL;
	r_ActivePower		: 	REAL;
	
	//Power
	r_ApparentPhasePower	: 	ARRAY[0..3] OF REAL;
	r_ReactivePhasePower	: 	ARRAY[0..3] OF REAL;
	r_ActivePhasePower		: 	ARRAY[0..3] OF REAL;

	//Energy Consumed
	r_EnergyConsumed	:	REAL;
	
	//Energy Delivered
	r_EnergySupplied	:	REAL;

	//currents
	r_Current			:	ARRAY[0..4] OF REAL;
	
	//THD
	r_THD				:	ARRAY[0..3] OF REAL;

	r_PowerFactor		:	ARRAY[0..3] OF REAL;
	
END_STRUCT
END_TYPE

// ---- POUs/Objects/PowerQualityMonitor/_Structs/ST_PowerMonitor_OutputField.TcDUT
TYPE ST_PowerMonitor_OutputField :
STRUCT
	e_ACrotationStatus	:	eACRotationState;
	r_Frequency			: 	REAL;
	
	r_PhaseVoltage		: 	ARRAY[0..3] OF REAL;
	r_LineVoltage		:	ARRAY[0..3] OF REAL;
	
		//Power
	r_ApparentPower		: 	REAL;
	r_ReactivePower		: 	REAL;
	r_ActivePower		: 	REAL;
	
	//Power
	r_ApparentPhasePower	: 	ARRAY[0..3] OF REAL;
	r_ReactivePhasePower	: 	ARRAY[0..3] OF REAL;
	r_ActivePhasePower		: 	ARRAY[0..3] OF REAL;

	//Energy Consumed
	r_EnergyConsumed	:	REAL;
	r_EnergySupplied	:	REAL;
	
	//currents
	r_Current			:	ARRAY[0..4] OF REAL;
	
	//THD
	r_THD				:	ARRAY[0..3] OF REAL;
	
	//VoltageUnbalance
	r_VoltageUnbalance	: 	ARRAY[0..3] OF REAL;

	r_PowerFactor		:	ARRAY[0..3] OF REAL;
	
	//PowerLock Currents, 3 fields of 4 measurements
	ar_PowerlockCurrents		: 	ARRAY [1..3] OF ARRAY[0..4] OF REAL;
END_STRUCT
END_TYPE

// ---- POUs/Objects/PowerStack/eNums/eNetcontactorState.TcDUT
{attribute 'qualified_only'}
{attribute 'strict'}
{attribute 'to_string'}
TYPE eNetcontactorState :
(
	Open 			:= 0,
	RightClosed		:= 1,
	LeftClosed		:= 2,
	Fault			:= 4
);
END_TYPE

// ---- POUs/Objects/PowerStack/eNums/eStatus.TcDUT
{attribute 'qualified_only'}
{attribute 'strict'}
{attribute 'to_string'}
TYPE eStatus :
(
	Init					:= 0,	// Not ready to do anything yet
	off						:= 1, 	// OFF MCCBs OPEN,
	idle					:= 2, 	// MCCB CLOSED, No modulation, Netcontactor CLOSED
	running					:= 3,	// MCCB CLOSED + Modulation, Netcontactor CLOSED
	ecorunning				:= 4,	// MCCB CLOSED + Modulation with only one out of two inverters, Netcontactor CLOSED
	fault					:= 5,	// FAULT STATE
	starting_master			:= 6, 	// Starting master
	starting_slave			:= 7,	// Starting slave
	Standby_GridSupply		:= 8, 	// POWERMODULE 1 + 2 off, Netcontactor Closed
	Standby_InternalSupply	:= 9,	// PowerModule 1 ON, powermodule 2 Off, Netcontactor OPEN
	shutdown				:= 10
);		
END_TYPE

// ---- POUs/Objects/PowerStack/st_Powerstack_get.TcDUT
TYPE ST_PowerStack_get :
STRUCT
	// READ
//	e_InverterMode					: eInverterModes;			//0=AFE, Micro, Island, transition
//	e_PowerMode						: ePowerModes;				//0=IsoChronous, 1= Droop
	r_VoltageDroop					: REAL;				
	r_FrequencyDroop				: REAL;
	r_NominalD7Voltage				: REAL; 
	r_NominalD7Frequency			: REAL; 
	r_ActivePower					: REAL; 
	r_ReactivePower					: REAL; 
	r_MaxChargePower				: REAL;
	r_MaxDischargePower				: REAL; 
	r_MaxCurrentAC					: REAL;
	r_PowerChangeRate				: REAL;
	r_ApparentPower					: REAL;
	r_CosPhi						: REAL;
	r_AcCurrent						: REAL;
	r_DCPower						: REAL;
	r_DCVoltage						: REAL;
	r_DCcurrent						: REAL;
	r_ACSupplyVoltage				: REAL;
	r_ACSupplyFrequency				: REAL;
	r_LoadPercentage				: REAL; //%
	r_RatedCurrent					: REAL;
	r_RatedPower					: REAL;
//	e_Status						: eStatus;
	e_NetContactorStatus			: eNetContactorState;
	
	b_CoolingRequest				: BOOL; //0=off, 1=on
	b_HVDCRequest					: BOOL; //0=off, 1=on
	//Temperature structure per powermodule toevoegen
//	Faults							: ST_PowerStackFaults;
	
END_STRUCT
END_TYPE

// ---- POUs/Objects/ProtectionSystems/FireDetection/eNums/eFireAlarmStatus.TcDUT
{attribute 'qualified_only'}
{attribute 'strict'}
TYPE eFireAlarmStatus :
(
	Error := 0,
	Normal := 1,
	Alarm := 2
);
END_TYPE

// ---- POUs/Objects/ProtectionSystems/FireDetection/eNums/eCOAlarmStatus.TcDUT
{attribute 'qualified_only'}
{attribute 'strict'}
TYPE eCOAlarmStatus :
(
	Error			:= 0,
	Normal 			:= 1,
	WarningLevel1 	:= 2,
	WarningLevel2 	:= 3,
	Alarm 			:= 4
);
END_TYPE

// ---- POUs/Objects/ProtectionSystems/FireDetection/Structs/ST_COInputData.TcDUT
TYPE ST_COInputData :
STRUCT
	w_Value				:	WORD;
	b_InputUnderrange 	: 	BOOL;
	b_InputOverrange	:	BOOL;
END_STRUCT
END_TYPE

// ---- POUs/Objects/ProtectionSystems/FireDetection/Structs/ST_FireDetectionGet.TcDUT
TYPE ST_FireDetectionGet :
STRUCT
	SmokeDetected		:	BOOL;					//-1 if inoperative.
	CODetectorValues 	:  	ARRAY[0..2] OF REAL;	//-1 if inoperative.
	
	Events	:	ST_FireSystem_Events;
END_STRUCT
END_TYPE

// ---- POUs/Objects/ProtectionSystems/FireDetection/Structs/ST_FireDetectionSet.TcDUT
TYPE ST_FireDetectionSet :
STRUCT
	b_SilenceSounder	:	BOOL; //only disables currently activated alarm.
	b_TestSounder		:	BOOL;
END_STRUCT
END_TYPE

// ---- POUs/Objects/ProtectionSystems/FireDetection/Structs/ST_FireSystem_Events.TcDUT
TYPE ST_FireSystem_Events :
STRUCT
	b_CODetFault		:	BOOL;
	b_CODetWarning1		:	BOOL;
	b_CODetWarning2		:	BOOL;
	b_CODetAlarm		:	BOOL;
	
	b_SmokeDetFault		:	BOOL;
	b_SmokeDetAlarm		:	BOOL;
	
	b_AlarmMuted		:	BOOL;
END_STRUCT
END_TYPE

// ---- POUs/Objects/ProtectionSystems/FireDetection/Structs/ST_SmokeDetIO.TcDUT
TYPE ST_SmokeDetIO :
STRUCT
	b_SmokeDetectorSignal_OK 	: BOOL;
	b_SmokeDetectorPower_OK 	: BOOL;
	b_SmokeDetectorShutdown		: BOOL;
END_STRUCT
END_TYPE

// ---- POUs/Objects/RouterData/Struct/dwtoreal.TcDUT
TYPE dwtoreal :
UNION
	Registers	:	ARRAY[1..2] OF WORD;
	dwordvalue	:	dword;
	realvalue	:	REAL;
END_UNION
END_TYPE

// ---- POUs/Objects/RouterData/Struct/eSMSStatus.TcDUT
{attribute 'qualified_only'}
{attribute 'strict'}
TYPE eSMSStatus :
(
	Idle 			:= 	0,
	NewMessage 		:= 	1,
	SendingMessage 	:= 	2,
	error			:=	3
);
END_TYPE

// ---- POUs/Objects/RouterData/Struct/st_Device.TcDUT
TYPE st_Device :
STRUCT
	SystemUptime	:	UDINT;	
	Temperature		:	REAL;
	RouterSerial	:	STRING(32);
END_STRUCT
END_TYPE

// ---- POUs/Objects/RouterData/Struct/st_GPS.TcDUT
TYPE st_GPS :
STRUCT
	Latitude 	: 	REAL;
	Longitude 	: 	REAL;
	FixTime 	: 	STRING(32);
	DateTime	:	STRING(32);
	Speed		:	REAL;
	SatCount	:	UINT;
	Accuracy	:	REAL;	
END_STRUCT
END_TYPE

// ---- POUs/Objects/RouterData/Struct/st_mobile.TcDUT
TYPE st_mobile :
STRUCT
	NetworkOperator				:	STRING(32);
	NetworkInfo					:	STRING(32);
	NetworkType					:	STRING(32);
	RSSI						:	DINT;
	ui_ActiveSim				:	UINT;
	ui_Sim1DataSendMonth		:	UINT;
	ui_Sim1DataReceivedMonth	:	UINT;
	ui_Sim2DataSendMonth		:	UINT;
	ui_Sim2DataReceivedMonth	:	UINT;
	s_EmergencySMSNumber		:	STRING(20);
	s_EmergencySMSDevName		:	STRING(8);
	st_LatestSMSMessage			:	STRING(80);
END_STRUCT
END_TYPE

// ---- POUs/Objects/RouterData/Struct/st_router_data.TcDUT
TYPE st_router_data :
STRUCT
	Device 		: 	st_Device;
	GPS			:	st_GPS;
	Mobile		:	st_mobile;
	e_SMSStatus : 	eSMSStatus;
	Events		:	st_TeltonikaEvents;
END_STRUCT
END_TYPE

// ---- POUs/Objects/RouterData/Struct/ST_Router_params.TcDUT
TYPE ST_Router_params :
STRUCT
	IP_TELTONIKA		: STRING(16) := '192.168.001.001';
	MBPort_TELTONIKA 	: UINT := 502;
	T_MBTimeout			: TIME := T#200MS;
	MinimumPhoneNumberLength	:	UINT := 10;
END_STRUCT
END_TYPE

// ---- POUs/Objects/RouterData/Struct/st_TeltonikaEvents.TcDUT
TYPE st_TeltonikaEvents :
STRUCT
	b_MBCommWarning		:	BOOL;
	b_MBCommError		:	BOOL;
	b_NoSimWarning		:	BOOL;
	b_NoNetworkWarning	: 	BOOL;
	b_noGPSFixWarning	:	BOOL;
	b_SMSNotSendError	:	BOOL; 
	b_NoSMSNumberAvailable	:	BOOL;
END_STRUCT
END_TYPE

// ---- POUs/System/_Structs/ST_SystemControl_FromSystem.TcDUT
{ attribute 'TcHmiSymbol.ShowRecursively' }

TYPE ST_SystemControl_FromSystem :
STRUCT
	b_modeSwitchEnable					: BOOL;
	
	safety								: ST_Safety_get;
	system								: ST_SystemControl_System;
	powerstack							: ST_Powerstack_get;
	powermonitor						: ST_PowerMonitor_get;
	ACswitchgear						: ST_ACSwitchgear_Get;
	neutraltransformer					: ST_NeutralTransformer_Get;
	battery								: st_MBMU_BatterySummary;
	protections							: ST_ProtectionSystems_get;
	peakshavebox						: ST_Peakshavebox_get;
	enclosure							: ST_Enclosure_get;
	internalpsu							: ST_InternalPowersupply_Get;
	DCswitchgear						: ST_DCSwitchgear_Get;
	PLC									: ST_plcstate_get;
	Properties							: ST_System_properties;
	//Cooling							
END_STRUCT
END_TYPE

// ---- POUs/System/_Structs/TempStructs/eCOAlarmStatus_1.TcDUT
{attribute 'qualified_only'}
{attribute 'strict'}
{attribute 'tostring'}
TYPE eCOAlarmStatus_1 :
(
	Error			:= 0,
	Normal 			:= 1,
	WarningLevel1 	:= 2,
	WarningLevel2 	:= 3,
	Alarm 			:= 4
);
END_TYPE

// ---- POUs/System/_Structs/TempStructs/eSmokeDetectAlarmStatus.TcDUT
{attribute 'qualified_only'}
{attribute 'strict'}
{attribute 'tostring'}
TYPE eSmokeDetectAlarmStatus :
(
	Error := 0,
	Normal := 1,
	Alarm := 2
);
END_TYPE

// ---- POUs/System/_Structs/TempStructs/eWago750495_ACDataID.TcDUT
{attribute 'qualified_only'}
{attribute 'strict'}
{attribute 'to_String'}
TYPE eWago750495_ACDataID :
(
	//only RMS and peak values are declared
	//Voltages
	VoltageL1N_RMS			:= 4,
	VoltageL2N_RMS 			:= 5,
	VoltageL3N_RMS			:= 6,
	VoltageL1L2_RMS			:= 31,
	VoltageL2L3_RMS 		:= 32,
	VoltageL3L1_RMS			:= 33,
	VoltageL1N_Peak 		:= 91,
	VoltageL2N_Peak 		:= 92,
	VoltageL3N_Peak 		:= 93,
	
	//Currents
	CurrentL1_RMS			:= 1,
	CurrentL2_RMS			:= 2,
	CurrentL3_RMS			:= 3,
	CurrentN_RMS			:= 97,
	CurrentL1_Peak			:= 94,
	CurrentL2_Peak			:= 95,
	CurrentL3_Peak			:= 96,
	                           
	//Power                    
	ActivePowerL1			:= 07,
	ActivePowerL2			:= 08,
	ActivePowerL3			:= 09,
	ReactivePowerL1			:= 10,
	ReactivePowerL2			:= 11,
	ReactivePowerL3			:= 12,
	ApparentPowerL1			:= 13,
	ApparentPowerL2			:= 14,
	ApparentPowerL3			:= 15,
	
	//Energy
	ActiveEnergyTotal			:= 73,
	ActiveEnergyImport			:= 74,
	ActiveEnergyExport			:= 75,
	ReactiveEnergyTotal			:= 85,
	ReactiveEnergyInductive		:= 86,
	AReactiveEnergyCapacitive	:= 87,
	
	//Frequency
	FrequencyL1				:= 16,
	FrequencyL2				:= 17,
	FrequencyL3				:= 18,
	                           
	//Phase Angle              
	PhaseAngleL1			:= 19,
	PhaseAngleL2			:= 20,
	PhaseAngleL3			:= 21,
	
	//PowerFactor
	PowerFactorL1			:= 25,
	PowerFactorL2			:= 26,
	PowerFactorL3			:= 27
) USINT;
END_TYPE

// ---- POUs/System/_Structs/TempStructs/eWago750495_HarmonicsDataID.TcDUT
{attribute 'qualified_only'}
{attribute 'strict'}
{attribute 'to_String'}
TYPE eWago750495_HarmonicsDataID :
(
	Current_RMS 		:= 001,
	Voltage_RMS 		:= 002,
	CurrentTHD			:= 003,
	VoltageTHD			:= 004
	
	//harmonics not declared for now
);
END_TYPE

// ---- POUs/System/_Structs/TempStructs/eWago750495_MeasureGroupID.TcDUT
{attribute 'qualified_only'}
{attribute 'strict'}
{attribute 'to_String'}
TYPE eWago750495_MeasureGroupID :
(
	ac := 10,
	harmonicsL1 := 20,
	harmonicsL2 := 21,
	harmonicsL3	:= 22
) USINT;
END_TYPE

// ---- POUs/System/_Structs/TempStructs/eWago750495_StatDataID.TcDUT
{attribute 'qualified_only'}
{attribute 'strict'}
TYPE eWago750495_StatDataID :
(
	Phase1 := 0,
	Phase2 := 1,
	Phase3 := 2,
	IOmodule:= 3
)USINT;
END_TYPE

// ---- POUs/System/_Structs/TempStructs/ST_ACSwitchgear_Get.TcDUT
TYPE ST_ACSwitchgear_Get :
STRUCT
	b_InputMCCBfb			: BOOL;
	b_InputMCCBShuntOK		: BOOL;	
	b_OutputMCCBfb			: BOOL;
	b_OutputMCCBShuntOK		: BOOL;
	b_CEEprefuseOK			: BOOL;
	b_InputSynchronizerfb	: BOOL;
	b_InputContactorfb		: BOOL;
	b_PENlinkfb				: BOOL;
	b_ExtIOSignal			: BOOL;
END_STRUCT
END_TYPE

// ---- POUs/System/_Structs/TempStructs/ST_CODetectors.TcDUT
TYPE ST_CODetectors :
STRUCT
	State 			: 	eCOAlarmStatus;
	b_CoValuesOK	: 	BOOL;
	Value 			:  	ARRAY[0..2] OF REAL;	//-1 if inoperative.
END_STRUCT
END_TYPE

// ---- POUs/System/_Structs/TempStructs/ST_DCSwitchgear_Get.TcDUT
TYPE ST_DCSwitchgear_Get :
STRUCT
	b_DCCouplingState				: BOOL;
	r_DCcouplingCurrent				: REAL;
END_STRUCT
END_TYPE

// ---- POUs/System/_Structs/TempStructs/ST_Enclosure_get.TcDUT
TYPE ST_Enclosure_get :
STRUCT
	climate				: REFERENCE TO ST_EnclosureClimate_Get;
	doors				: REFERENCE TO ST_DoorsNLocks_events;
	ledstrip			: REFERENCE TO ST_Ledstrip_events;
END_STRUCT
END_TYPE

// ---- POUs/System/_Structs/TempStructs/ST_FireDetection_get.TcDUT
TYPE ST_FireDetection_get :
STRUCT
	SmokeDetectors : ST_SmokeDetectors;
	CODetectors	:	ST_CODetectors;
	
	Events	:	ST_FireSystem_Events;
END_STRUCT
END_TYPE

// ---- POUs/System/_Structs/TempStructs/ST_FireDetection_get_1.TcDUT
TYPE ST_FireDetection_get_1 :
STRUCT
	SmokeDetectors : ST_SmokeDetectors;
	CODetectors	:	ST_CODetectors;
	
	Events	:	ST_FireSystem_Events;
END_STRUCT
END_TYPE

// ---- POUs/System/_Structs/TempStructs/ST_FireDetection_set.TcDUT
TYPE ST_FireDetection_set :
STRUCT
	SilenceSounder	:	BOOL; //only disables currently activated alarm.
	TestSounder		:	BOOL;
END_STRUCT
END_TYPE

// ---- POUs/System/_Structs/TempStructs/ST_FireSystem_Events_1.TcDUT
TYPE ST_FireSystem_Events_1 :
STRUCT
	CODetFault		:	BOOL;
	CODetWarning	:	BOOL;
	CODetAlarm		:	BOOL;
	SmokeDetFault	:	BOOL;
	SmokeDetAlarm	:	BOOL;
	AlarmMuted		:	BOOL;
END_STRUCT
END_TYPE

// ---- POUs/System/_Structs/TempStructs/ST_FireSystem_Events_2.TcDUT
TYPE ST_FireSystem_Events_2 :
STRUCT
	CODetFault		:	BOOL;
	CODetWarning	:	BOOL;
	CODetAlarm		:	BOOL;
	SmokeDetFault	:	BOOL;
	SmokeDetAlarm	:	BOOL;
	AlarmMuted		:	BOOL;
END_STRUCT
END_TYPE

// ---- POUs/System/_Structs/TempStructs/ST_InsulationMonitor_get.TcDUT
TYPE ST_InsulationMonitor_get :
STRUCT
	b_Enabled							: BOOL;	
	b_PENlinkNotDetected				: BOOL;
	b_Warning							: BOOL;
END_STRUCT
END_TYPE

// ---- POUs/System/_Structs/TempStructs/ST_NeutralTransformer_Get.TcDUT
TYPE ST_NeutralTransformer_Get :
STRUCT
	r_TemperaturePhase							: ARRAY [0..6] OF REAL;
	r_Powerload									: REAL;
	events										: ST_NeutralTransformer_events;
END_STRUCT
END_TYPE

// ---- POUs/System/_Structs/TempStructs/ST_OvercurrentProtection_get.TcDUT
TYPE ST_OvercurrentProtection_get :
STRUCT
	//Overcurrent Powerlocks
	b_OutputWarning						: BOOL;
	b_InputWarning						: BOOL;
	b_OutputAlarm						: BOOL;
	b_InputAlarm						: BOOL;
	r_PeakCurrent						: REAL;
	t_PeakCurrentDuration				: TIME;
	s_locationPeak						: STRING;
	
	Events								: ST_OvercurrentProtection_events;
END_STRUCT
END_TYPE

// ---- POUs/System/_Structs/TempStructs/ST_PeakShaveBox_Get.TcDUT
TYPE ST_PeakShaveBox_Get :
STRUCT
	Powermonitor		: ST_Wago750495_Get;
	Buscoupler			: ST_Wago750354_get;
END_STRUCT
END_TYPE

// ---- POUs/System/_Structs/TempStructs/ST_PLCstate_get.TcDUT
TYPE ST_PLCstate_get :
STRUCT
	r_CPUload		: REAL;
	e_ProfinetState	: eNetcomState;
	e_EthercatState	: eNetcomState;
END_STRUCT
END_TYPE

// ---- POUs/System/_Structs/TempStructs/ST_ProtectionSystems_get.TcDUT
TYPE ST_ProtectionSystems_get :
STRUCT
	//Fire Detection System
	FireDetection						: REFERENCE TO ST_Firedetection_get;
	
	//InsulationMonitor
	Insulation							: REFERENCE TO ST_InsulationMonitor_get;
	
	//MRCDB
	MRCDB								: REFERENCE TO ST_ResidualCurrentMonitor_get;
	
	//Surge protection
	Surge								: REFERENCE TO ST_SurgeProtection_get;
	
	//Overcurrent protection
	OvercurrentProtection				: REFERENCE TO ST_OverCurrentProtection_Get;
	
END_STRUCT
END_TYPE

// ---- POUs/System/_Structs/TempStructs/ST_ResidualCurrentMonitor_get.TcDUT
TYPE ST_ResidualCurrentMonitor_get :
STRUCT
	b_prewarning			: BOOL;
END_STRUCT
END_TYPE

// ---- POUs/System/_Structs/TempStructs/ST_Safety_get.TcDUT
TYPE ST_Safety_get :
STRUCT
	b_SafetyOK					: BOOL;
	b_EstopChannelAOK			: BOOL;		
	b_EstopChannelBOK			: BOOL;		
	b_InsulationMonitorOK		: BOOL;	
	b_MRCDBOK					: BOOL;	
	b_InverterDoorOK            : BOOL;
	b_ZptOK				        : BOOL;
END_STRUCT
END_TYPE

// ---- POUs/System/_Structs/TempStructs/ST_Safety_get_1.TcDUT
TYPE ST_Safety_get_1 :
STRUCT
	b_SafetyOK					: BOOL;
	b_EstopChannelAOK			: BOOL;		
	b_EstopChannelBOK			: BOOL;		
	b_InsulationMonitorOK		: BOOL;	
	b_MRCDBOK					: BOOL;	
	b_InverterDoorOK            : BOOL;
	b_ZptOK				        : BOOL;
END_STRUCT
END_TYPE

// ---- POUs/System/_Structs/TempStructs/ST_SmokeDetectors.TcDUT
TYPE ST_SmokeDetectors :
STRUCT
	State : eSmokeDetectAlarmStatus;
END_STRUCT
END_TYPE

// ---- POUs/System/_Structs/TempStructs/ST_SmokeDetIO_1.TcDUT
TYPE ST_SmokeDetIO_1 :
STRUCT
	SmokeDetectorSignal_OK 	: BOOL;
	SmokeDetectorPower_OK 	: BOOL;
	SmokeDetectorShutdown	: BOOL;
END_STRUCT
END_TYPE

// ---- POUs/System/_Structs/TempStructs/ST_Surgeprotection_get.TcDUT
TYPE ST_Surgeprotection_get :
STRUCT
	b_Type12_OK				: BOOL;
	b_Type3_OK				: BOOL;			
END_STRUCT
END_TYPE

// ---- POUs/System/_Structs/TempStructs/ST_SystemControl_System.TcDUT
TYPE ST_SystemControl_System :
STRUCT
	
	//Statuss
	e_State						: eSystemState; //0:Idle, 1: Stand-by, 2:Conditioning, 3:Dry-Cycle, 4: Running, 5: Charging only, 6: Discharging only, 7: Stopped 8:Fault, 10: Reset
	e_EarthingSystem			: eEarthingSystems; //0: Unknown, 1: TN-S, 2: TN-C, 3: IT.
	PowerController				: ST_PowerControl_get;
	
	
	
	//LIMITS
	r_Pmin						: REAL ;
	r_Pmax						: REAL ;
	r_QMin						: REAL ;
	r_QMax						: REAL ;
	r_AcCurrentMax				: REAL := 520;
	
END_STRUCT
END_TYPE

// ---- POUs/System/_Structs/TempStructs/ST_System_Properties.TcDUT
TYPE ST_System_Properties :
STRUCT
	r_RatedActivePower		: REAL;
	r_RatedApparentPower	: REAL;
	r_RatedCurrent			: REAL;
	r_RatedEnergyCapacity	: REAL;
	r_SelfdischargeRate		: REAL;
	r_RatedSoCMax			: REAL;
	r_RatedSocMin			: REAL;
	s_ManufacturerModel		: STRING := 'e-PU10';
	s_Options				: STRING;
	s_SerialNumber			: STRING;
	s_VersionNumber			: STRING;
END_STRUCT
END_TYPE

// ---- POUs/System/_Structs/TempStructs/ST_Wago750354_get.TcDUT
TYPE ST_Wago750354_get :
STRUCT
	b_SlaveReady							: BOOL;
END_STRUCT
END_TYPE

// ---- POUs/System/_Structs/TempStructs/ST_Wago750495_Data.TcDUT
TYPE ST_Wago750495_Data :
STRUCT
	//Voltages
	r_VoltageL1N_RMS				: REAL;
	r_VoltageL2N_RMS 				: REAL;
	r_VoltageL3N_RMS				: REAL;
	r_VoltageL1L2_RMS				: REAL;
	r_VoltageL2L3_RMS 				: REAL;
	r_VoltageL3L1_RMS				: REAL;
	r_VoltageL1N_Peak 				: REAL;
	r_VoltageL2N_Peak 				: REAL;
	r_VoltageL3N_Peak 				: REAL;
	                            	      
	//Currents                  	      
	r_CurrentL1_RMS					: REAL;
	r_CurrentL2_RMS					: REAL;
	r_CurrentL3_RMS					: REAL;
	r_CurrentN_RMS					: REAL;
	r_CurrentL1_Peak				: REAL;
	r_CurrentL2_Peak				: REAL;
	r_CurrentL3_Peak				: REAL;
	                            	      
	//Power                     	      
	r_ActivePowerL1					: REAL;
	r_ActivePowerL2					: REAL;
	r_ActivePowerL3					: REAL;
	r_ReactivePowerL1				: REAL;
	r_ReactivePowerL2				: REAL;
	r_ReactivePowerL3				: REAL;
	r_ApparentPowerL1				: REAL;
	r_ApparentPowerL2				: REAL;
	r_ApparentPowerL3				: REAL;
	
	//Energy
	r_ActiveEnergyTotal				: REAL;
	r_ActiveEnergyImport			: REAL;
	r_ActiveEnergyExport			: REAL;
	r_ReactiveEnergyTotal			: REAL;
	r_ReactiveEnergyInductive		: REAL;
	r_AReactiveEnergyCapacitive		: REAL;
	
	//Frequency
	r_FrequencyL1					: REAL;
	r_FrequencyL2					: REAL;
	r_FrequencyL3					: REAL;
	                        		      
	//Phase Angle           		      
	r_PhaseAngleL1					: REAL;
	r_PhaseAngleL2					: REAL;
	r_PhaseAngleL3					: REAL;
	                        		      
	//PowerFactor           		      
	r_PowerFactorL1					: REAL;
	r_PowerFactorL2					: REAL;
	r_PowerFactorL3					: REAL;
	
	
END_STRUCT
END_TYPE

// ---- POUs/System/_Structs/TempStructs/ST_Wago750495_ExtStatusWord.TcDUT
TYPE ST_Wago750495_ExtStatusWord :
STRUCT
	b_IncreasedMeasErr			: BOOL; //Stat 1 query L1,L2,L3:: increase measurement error of selected phase
	b_CurrentClipping			: BOOL; //Stat 2 query L1,L2,L3:: current out of measurable range of selected phase
	b_VoltageClipping			: BOOL; //Stat 3 query L1,L2,L3:: voltage out of measurable range of selected phase
	b_NoZeroCrossings			: BOOL; //Stat 4 query L1,L2,L3:: Zero Crossings missing of selected phase
	b_OverCurrent				: BOOL; //Stat 5 query L1,L2,L3:: Overcurrent of selected phase
	b_OverVoltage				: BOOL; //Stat 6- query L1,L2,L3: OverVoltage of selected phase.
	b_RotaryField				: BOOL; //Stat 6- query IO: 0:Clockwise, 1: counterclockwise
	b_UnderVoltage				: BOOL; //Stat 7- query L1,L2,L3: UnderVoltage of selected phase

END_STRUCT
END_TYPE

// ---- POUs/System/_Structs/TempStructs/ST_Wago750495_Get.TcDUT
TYPE ST_Wago750495_Get :
STRUCT
	StatusWord				: ST_Wago750495_StatusWord;
	ExtStatusWord			: ST_Wago750495_ExtStatusWord;
	Data					: ST_Wago750495_Data;
END_STRUCT
END_TYPE

// ---- POUs/System/_Structs/TempStructs/ST_Wago750495_Set.TcDUT
TYPE ST_Wago750495_Set :
STRUCT
	b_EnableRegisterComm		: BOOL;
	e_statusQuery				: eWago750495_StatDataID; //0: status L1, 1: status L2, 2: Status L3, 3: Status IO Module			
END_STRUCT
END_TYPE

// ---- POUs/System/_Structs/TempStructs/ST_Wago750495_StatusWord.TcDUT
TYPE ST_Wago750495_StatusWord :
STRUCT
	b_ComFb						: BOOL; // 0: process Data, 1: Register Data
	b_Error						: BOOL; // 0: OK, 1: Error
	b_Error_IO					: BOOL; // 0: OK, 1: Error
	b_Error_L3					: BOOL; // 0: OK, 1: Error
	b_Error_L2					: BOOL; // 0: OK, 1: Error
	b_Error_L1					: BOOL; // 0: OK, 1: Error
	e_StatIDfb					: eWago750495_StatDataID;
	b_Warning					: BOOL; // 0: OK, 1: Transient reaction measured value collection active
	b_Cal						: BOOL; // 0: Measurement Mode, 1: Calibration Mode
	b_Over_1					: BOOL; // 0: OK, 1: Out Of Range
	b_Over_2					: BOOL; // 0: OK, 1: Out Of Range
	b_Over_3					: BOOL; // 0: OK, 1: Out Of Range
	b_Over_4					: BOOL; // 0: OK, 1: Out Of Range
	e_GroupID					: eWago750495_MeasureGroupID;

END_STRUCT
END_TYPE

// ---- GVLs/Config.TcGVL
{attribute 'qualified_only'}
VAR_GLOBAL CONSTANT
	b_DoublePowerModule				: BOOL := FALSE;
	b_PeakshaverBoxEnable			: BOOL := TRUE;
	b_NeutralTransformer			: BOOL := TRUE;
	
	//Netcontactor
	b_AutomaticACrotation			: BOOL := TRUE;
	b_DoubleHeatpump: BOOL := FALSE;
	
	IP_BMS	:	STRING(16) := '192.168.1.61';
	MBPort_BMS : UINT := 502;
	
	IP_JANITZA: STRING(16) := '192.168.1.10';
	MBPort_Janitza : UINT := 502;

	IP_Teltonika: STRING(16) := '192.168.1.1';
	MBPort_Teltonika : UINT := 502;

	

END_VAR

// ---- GVLs/GVL.TcGVL
{attribute 'qualified_only'}
VAR_GLOBAL
	{define InputField}
	{define ThirdOutputField}
	s_SystemTime				: STRING;
	s_SystemDate				: STRING;

	b_initCycle							: BOOL := TRUE;
	b_reset								: BOOL;
	
	
	//error variables
	b_WarningActive						: BOOL;
	b_NormalShutdownActive				: BOOL;
	b_QuickshutdownActive				: BOOL;
	b_EmergencyShutdownActive			: BOOL;	
	
	
END_VAR

VAR_GLOBAL CONSTANT
	t_HMIUpdateTime						: TIME:= T#500MS;
END_VAR

// ---- POUs/Objects/CoolingSystem/CoolingSystemParams.TcGVL
{attribute 'qualified_only'}
VAR_GLOBAL CONSTANT
	
	//Main cooling regulation settings
	PIDControlLimitMax: REAL := 10.0;
	PIDControlLimitMin: REAL := 10.0;
	PIDControlKfactor: 	REAL := 0.1;
	PIDControlTn: 		TIME := T#1000MS;//Integral coefficient
	PIDControlTv: 		TIME := T#0MS;//Derivative coefficient 
	PIDControlTd: 		TIME := T#60S;//Damping time 
	PIDLoopTime:		TIME := T#1000MS;//
	
	BattGoalTemp		: 	REAL := 18.0;
	CoolantFullPowerTemperatureOffset: REAL := 1.5;
	

	EnclosureActiveTempMin: REAL := 10.0;
	EnclosureActiveTempMax: REAL := 40.0;
	
	//setpoints for enclosure dehum
	EnclosureDewPointGoal: REAL := 10.0;
	EnclosureDewPointHysteresis: REAL := 2.0;
	
	EnclosureIdleTempMin: REAL := 10.0;
	EnclosureIdleTempMax: REAL := 30.0;
	
	BatteryIdleTempMin	:	REAL	:=	15.0;
	BatteryIdleTempMax	:	REAL	:=	20.0;
	
	HeatpumpInitSettings	: WORD := 0;
	DoubleHeatpump			: BOOL := FALSE;
	
	//max temperature of the inverter components before cooling system can shutdown
	EMSTOPInverterIdleShutdownTemp 		: REAL := 40;
	//max temperature of the Battery components before cooling system can shutdown
	EMSTOPBatteryShutdownTemp			: REAL := 25; 
	
	// Minimum base coolant pressure
	MinimumSystemBasePressureWarningLevel	:	REAL :=	1.5;
	MinimumSystemBasePressureErrorLevel		:	REAL :=	1;
	// Minimum cooling system pressure increase with 24V pump running
	StartupPumpMinimumPressure	:	REAL	:= 0.2;
	// minimum cooling system pressure increase with main pump running
	MainPumpMinimumPressure				:	REAL	:= 0.5;
	
	
	MaximumValveOperatingTime	:	TIME := TIME#1000MS;


END_VAR

// ---- POUs/Objects/InternalPowerSupply/IPSParams.TcGVL
{attribute 'qualified_only'}
VAR_GLOBAL CONSTANT
	IntZPTStartupDelay: TIME := TIME#100MS;
	ACStartupDelay : TIME := TIME#100MS;
	DCPSU_StartupDelay: TIME := TIME#500MS;
	ACPSU_StartupDelay: TIME := TIME#500MS;
	//trigger level before Battery low error is issued. 
	//UPS battery dangerously low
	usi_UPSBattLowErrorSOC		:	USINT 	:= 20;
	//UPS charging request was apparently denied. System should shutdown? 
	usi_UPSBattLowwarningSOC	:	USINT 	:= 40;
	//trigger level before Battery low warning is issued and UPS charging is requested from Internal power supply
	usi_UPSBattLowinfoSOC		:	USINT	:= 60;	
	//r_SOC level at which UPS charging is no longer requested so HVDC can be shutdown.
	usi_UPSBattOKSOC 			:	USINT	:= 90;
END_VAR

// ---- POUs/Objects/PowerQualityMonitor/FB_Janitza_UMG801/PowerMeterConfig.TcGVL
{attribute 'qualified_only'}
VAR_GLOBAL CONSTANT
	IP_JANITZA: STRING(16) := '192.168.1.52';
	MBPort_Janitza : UINT := 502;
	
	b_ThirdOutputFieldAvailable	: BOOL 	:=	TRUE;
	b_InputFieldsAvailable		: BOOL	:=	TRUE;
END_VAR

// ---- POUs/MAIN.TcPOU
PROGRAM MAIN
VAR

//	PQMeter : FB_PowerQualityMonitoring;
	//FireSystem	: FB_FireDetection;
//	Data AT %I* : BYTE;
//	IPS	:	FB_InternalPowerSupply;
//	BMS: FB_BMS;
	
	ACPowerStatus 	: 	BOOL;
	MBFree			:	BOOL;
	Router	:	FB_Teltonika;
	
	MessageArray	:	ARRAY[1..3] OF STRING(75) := ['message1', 'Message2', 'Message3'];
	
//	CS	:	FB_CoolingSystem;

	//PN	:	FB_PNController;
	
	//HP	:	fb_HEATPUMPSYSTEM;
	
	by_PSCoolingPowerMode	:	BYTE := 0;
	by_setCooling			:	BYTE := 0;
	b_InverterRunning		:	BOOL := FALSE;
	r_InverterTemperature	: 	REAL := 20.0;
	r_InverterPowerLevel	: 	REAL := 0;
	r_CMSTemperature		: 	REAL := 20.0;
	b_24V_Available			:  	BOOL := FALSE;
	b_400v_available		: 	BOOL := FALSE;
	r_BMSAverageBattTemp	:	REAL := 20.0;
	r_BMSMaxBattTemp		: 	REAL := 20.0;
	r_EnclosureHumidity		: 	REAL := 20.0;
	r_EnclosureTemperature	: 	REAL := 20.0;
	
	//PNData AT %I*	:	WORD;
	
//	OperatingPoint	:	st_OperatingPoint;
	
	EMSTOPActive	:	BOOL;
	ResetActive		:	BOOL;
	(*
	MBTestInput			AT %I* :	ARRAY[0..3] OF WORD;
	MBTestOutput		AT %Q* :	ARRAY[0..3] OF WORD;
	
	SingleMBTestInput		AT %I* :	WORD;
	SingleMBTestOutput		AT %Q* :	WORD;
	
	HeartbeatIn		AT %I*	:	UINT;
	HeartbeatOut	AT %Q*	:	UINT	:= 0;
	
	SlaveHBin		AT %I*	:	UINT;
	SlaveHBOut		AT %Q*	:	UINT;
	*)
	HeartBeatTimer : TON := (Pt := T#1S);

	
	TestIn	AT %I* : ARRAY[1..7] OF BYTE;
	TestOut	AT %Q* : ARRAY[1..7] OF BYTE;

	TestInreg	AT %I* : ARRAY[1..10] OF WORD;
	TestOutreg	AT %Q* : ARRAY[1..10] OF WORD;
	
	MBTestOut 		AT %Q* :	WORD;
	MBTestin		AT %I* :	WORD;
	startConversion		: 	BOOL;
	TestString			:	STRING(20) := '0650749712';
	TestVar				:	BOOL; 
	
	GeneralOut			AT %Q* : ARRAY[1..11] OF WORD;
	GeneralIn			AT %I* : ARRAY[1..2] OF WORD;
	BMSOut				AT %Q* : ARRAY[1..17] OF WORD;
	BMSIn				AT %I* : ARRAY[1..2] OF WORD;
	OutputFieldOut		AT %Q* : ARRAY[1..20] OF WORD;
	InputFieldOut		AT %Q* : ARRAY[1..20] OF WORD;
	InputFieldIn		AT %I* : ARRAY[1..9] OF WORD;
	PowerStackOut		AT %Q* : ARRAY[1..17] OF WORD;
	PowerstackIn		AT %I* : ARRAY[1..15] OF WORD;
	PSBOut				AT %Q* : ARRAY[1..16] OF WORD;
	PSBIn				AT %I* : ARRAY[1..5] OF WORD;	
	ZPTOut				AT %Q* : ARRAY[1..6] OF WORD;
END_VAR

VAR
	LedStripSFC	:	UpdateSFC;
END_VAR

// Ik heb hier iets toegevoegd
//FireSystem();//TestSounder:=False);

//PQMeter();
//Router();
//IPS();
//extratje in main branch
(*
CS(	by_setCooling			:=	by_setCooling,
	b_InverterRunning 		:= 	b_InverterRunning,
	by_PSCoolingPowerMode	:=	by_PSCoolingPowerMode,
	r_InverterTemperature	:=	r_InverterTemperature,
	r_InverterPowerLevel	:=	r_InverterPowerLevel,
	r_CMSTemperature		:=	r_CMSTemperature,
	b_24V_Available			:=	b_24V_Available,
	b_400v_available		:=	b_400v_available,
	IPSDemand 				:= ips.Set.CoolingSystemPowerDemand,
	r_BMSAverageBattTemp	:=	r_BMSAverageBattTemp,
	r_BMSMaxBattTemp		:=	r_BMSMaxBattTemp,
	r_EnclosureHumidity		:=	r_EnclosureHumidity,
	r_EnclosureTemperature	:=	r_EnclosureTemperature
	);

	IF ResetActive THEN
		CS.Reset();
	END_IF

	IF //CS.Get.Events.b_BattLoopValveStuck OR
		CS.Get.Events.b_CoolingLoopIdlePressureError OR
		CS.Get.Events.b_InverterCoolingLoopError OR
		CS.Get.Events.b_CoolingSystemFuseFailure OR
		//CS.Get.Events.b_FancoilLoopValveStuck OR
		CS.Get.Events.b_HeatPumpError then
		//CS.Get.Events.b_InverterLoopValveStuck THEN
		CS.EMSTOP();
		END_IF;

//hp(b_EnablePower := ACPowerStatus);
//hp.WriteSetpoint(OperatingMode := OperatingPoint.OperatingMode, SetPoint := OperatingPoint.Setpoint);

//ReadDataTimer(in := NOT ReadDataTimer.Q);
//hp(ACPowerStatus:=ACPowerStatus, MBFree:=ReadDataTimer.q);
*)	
	
//BMS();

IF TRUE THEN
	ACPowerStatus := TRUE;
END_IF
(*
IF startConversion THEN
	TestVar := router.SetSMSNumber(TestString);
	startConversion := FALSE;
END_IF

//Router();
Router(s_message := MessageArray);
HeartBeatTimer(in:= NOT HeartBeatTimer.Q);

//MBTestOutput[0] := SingleMBTestInput;

IF HeartBeatTimer.Q THEN
	extTestOut[1] := extTestOut[1] + 1;
END_IF

extTestOut[2] := extTestOut[1]-1;
extTestOut[3] := extTestOut[2]-1;
extTestOut[4] := extTestOut[3]-1;
extTestOut[5] := extTestOut[4]-1;
extTestOut[6] := extTestOut[5]-1;

extTestIn[1];
extTestIn[2];
extTestIn[3];
extTestIn[4];
*)

//MBTestOut := MBTestin;
//TestOutreg[1] := TestInreg[1];
//TestOut := TestIn;


LedStripSFC();

//changeadded

END_PROGRAM

// ---- POUs/Objects/RouterData/FB_Teltonika.TcPOU
FUNCTION_BLOCK FB_Teltonika
VAR
	stRouterParams : st_router_params;
	realconverter : dwtoreal;
	w_SendSMS: WORD;
END_VAR
VAR_OUTPUT
	Get	:	st_router_data;
END_VAR
VAR
	MBRead			: 	FB_MBReadRegs;
	MBWrite			:	FB_MBWriteRegs;
	MBSingleWrite	:	FB_MBWriteSingleReg;
	
	arw_DataBuffer		: 	ARRAY[0..62] OF word;
	st_WriteSMSData		:	STRING(20);

	ar_SMSData			:	ARRAY[0..89] OF WORD;
	ar_ReadSMSData		:	ARRAY[0..89] OF WORD;

	
	ton_GetDataTimer				:	TON := (PT := TIME#1000MS);

	
	ftrig_TransmissionDone	:	F_trig;
	
	ui_MBRetryCount			:	UINT;
	ui_SMSRetryCounter	:	UINT;
		
	ui_ForCounter	:	UINT;
	ui_MessageCounter	:	UINT;
	b_busy: BOOL;
	b_CommError: BOOL;
	udi_errid: UDINT;
	udi_cbread: UDINT;
	
END_VAR


VAR_IN_OUT
	s_Message	:	ARRAY[*] OF STRING(75);
END_VAR

ton_GetDataTimer(IN:=NOT ton_GetDataTimer.Q);

ReadDataSFC();

get.Events.b_MBCommWarning := ui_MBRetryCount > 5;
IF ui_MBRetryCount > 50 THEN
	get.Events.b_MBCommError := TRUE;
END_IF

ACTION aCheckAlarmMessages:

IF get.e_SMSStatus = eSMSStatus.Idle OR get.e_SMSStatus = eSMSStatus.error THEN
	//skip through message array until non_empty value or the end of the list is found 
	WHILE (s_Message[ui_MessageCounter] = '') AND (ui_MessageCounter < UPPER_BOUND(s_message, 1)) DO
		ui_MessageCounter := ui_MessageCounter + 1;
	END_WHILE
	
	IF (s_Message[ui_MessageCounter] <> '') THEN
		CreateMessage(s_Message[ui_MessageCounter]);	//check for valid message
		get.e_SMSStatus := eSMSStatus.NewMessage;
		s_Message[ui_MessageCounter] := '';
	END_IF
	
	IF ui_MessageCounter >= UPPER_BOUND(s_message, 1) THEN
		ui_MessageCounter := DINT_TO_UINT(LOWER_BOUND(s_message, 1)); 
	END_IF
END_IF
END_ACTION

ACTION aNetworkinfo:
MBRead(
	sIPAddr := stRouterparams.IP_TELTONIKA,
	nTCPPort := stRouterparams.MBPort_TELTONIKA,
	nUnitID := 1,
	nMBAddr := 103,
	nQuantity := 32,//*2,
	cbLength := SIZEOF(arw_DataBuffer),
	pDestAddr := ADR(arw_DataBuffer),
	bExecute := ton_GetDataTimer.Q,
	bBusy => b_busy,
	bError => b_CommError,
	nErrId => udi_errid,
	cbRead => udi_cbread,
	tTimeout := stRouterparams.T_MBTimeout
);

ftrig_TransmissionDone(clk := b_busy);

IF ftrig_TransmissionDone.q THEN
	IF NOT b_CommError THEN
		FOR ui_ForCounter := 0 TO 31 DO
			arw_DataBuffer[ui_ForCounter] := be16_TO_HOST(arw_DataBuffer[ui_ForCounter]);
		END_FOR
		
		MEMCPY(ADR(Get.Mobile.NetworkInfo),  ADR(arw_DataBuffer[0]), 32);
		MEMCPY(ADR(Get.Mobile.NetworkType),  ADR(arw_DataBuffer[16]), 32);
		ui_MBRetryCount := 0;
		sfctip := TRUE;
	ELSE
		ui_MBRetryCount := ui_MBRetryCount + 1;
		sfctip := TRUE;
	END_IF
END_IF
END_ACTION

ACTION aReadActiveSim:

MBRead(
	sIPAddr := stRouterparams.IP_TELTONIKA,
	nTCPPort := stRouterparams.MBPort_TELTONIKA,
	nUnitID := 1,
	nMBAddr := 205,
	nQuantity := 1,//*2,
	cbLength := SIZEOF(arw_DataBuffer),
	pDestAddr := ADR(arw_DataBuffer),
	bExecute := ton_GetDataTimer.Q,
	bBusy => b_busy,
	bError => b_CommError,
	nErrId => udi_errid,
	cbRead => udi_cbread,
	tTimeout := stRouterparams.T_MBTimeout
);

ftrig_TransmissionDone(clk := b_busy);

IF ftrig_TransmissionDone.q THEN
	IF NOT b_CommError THEN
	
		Get.Mobile.ui_ActiveSim := arw_DataBuffer[0];
	
		ui_MBRetryCount := 0;
		sfctip := TRUE;
	ELSE
		ui_MBRetryCount := ui_MBRetryCount + 1;
		sfctip := TRUE;
	END_IF
END_IF
END_ACTION

ACTION aReadDataUsageSim1:

MBRead(
	sIPAddr := stRouterparams.IP_TELTONIKA,
	nTCPPort := stRouterparams.MBPort_TELTONIKA,
	nUnitID := 1,
	nMBAddr := 193,
	nQuantity := 4,//*2,
	cbLength := SIZEOF(arw_DataBuffer),
	pDestAddr := ADR(arw_DataBuffer),
	bExecute := ton_GetDataTimer.Q,
	bBusy => b_busy,
	bError => b_CommError,
	nErrId => udi_errid,
	cbRead => udi_cbread,
	tTimeout := stRouterparams.T_MBTimeout
);

ftrig_TransmissionDone(clk := b_busy);

IF ftrig_TransmissionDone.q THEN
	IF NOT b_CommError THEN
	
		MEMCPY(ADR(Get.Mobile.ui_Sim1DataReceivedMonth)+2, ADR(arw_DataBuffer[0]), 2);
		MEMCPY(ADR(Get.Mobile.ui_Sim1DataReceivedMonth), ADR(arw_DataBuffer[1]), 2);
		
		MEMCPY(ADR(Get.Mobile.ui_Sim1DataSendMonth)+2, ADR(arw_DataBuffer[2]), 2);
		MEMCPY(ADR(Get.Mobile.ui_Sim1DataSendMonth), ADR(arw_DataBuffer[3]), 2);	
	
		ui_MBRetryCount := 0;
		sfctip := TRUE;
	ELSE
		ui_MBRetryCount := ui_MBRetryCount + 1;
		sfctip := TRUE;
	END_IF
END_IF
END_ACTION

ACTION aReadDataUsageSim2:

MBRead(
	sIPAddr := stRouterparams.IP_TELTONIKA,
	nTCPPort := stRouterparams.MBPort_TELTONIKA,
	nUnitID := 1,
	nMBAddr := 308,
	nQuantity := 4,//*2,
	cbLength := SIZEOF(arw_DataBuffer),
	pDestAddr := ADR(arw_DataBuffer),
	bExecute := ton_GetDataTimer.Q,
	bBusy => b_busy,
	bError => b_CommError,
	nErrId => udi_errid,
	cbRead => udi_cbread,
	tTimeout := stRouterparams.T_MBTimeout
);

ftrig_TransmissionDone(clk := b_busy);

IF ftrig_TransmissionDone.q THEN
	IF NOT b_CommError THEN
	
		MEMCPY(ADR(Get.Mobile.ui_Sim2DataReceivedMonth)+2, ADR(arw_DataBuffer[0]), 2);
		MEMCPY(ADR(Get.Mobile.ui_Sim2DataReceivedMonth), ADR(arw_DataBuffer[1]), 2);
		
		MEMCPY(ADR(Get.Mobile.ui_Sim2DataSendMonth)+2, ADR(arw_DataBuffer[2]), 2);
		MEMCPY(ADR(Get.Mobile.ui_Sim2DataSendMonth), ADR(arw_DataBuffer[3]), 2);	
	
		ui_MBRetryCount := 0;
		sfctip := TRUE;
	ELSE
		ui_MBRetryCount := ui_MBRetryCount + 1;
		sfctip := TRUE;
	END_IF
END_IF
END_ACTION

ACTION AReadGeneral:

MBRead(
	sIPAddr := stRouterparams.IP_TELTONIKA,
	nTCPPort := stRouterparams.MBPort_TELTONIKA,
	nUnitID := 1,
	nMBAddr := 1,
	nQuantity := 6,//*2,
	cbLength := SIZEOF(arw_DataBuffer),
	pDestAddr := ADR(arw_DataBuffer),
	bExecute := ton_GetDataTimer.Q,
	bBusy => b_busy,
	bError => b_CommError,
	nErrId => udi_errid,
	cbRead => udi_cbread,
	tTimeout := stRouterparams.T_MBTimeout
);

ftrig_TransmissionDone(clk := b_busy);

IF ftrig_TransmissionDone.q THEN
	IF NOT b_CommError THEN
		
		get.Device.SystemUptime :=	SHL(	WORD_TO_UDINT(	arw_DataBuffer[0]),16)	+	arw_DataBuffer[1];
		MEMCPY(ADR(Get.Mobile.RSSI)+2,  ADR(arw_DataBuffer[2]), 2);
		MEMCPY(ADR(Get.Mobile.RSSI),  ADR(arw_DataBuffer[3]), 2);

		//MEMCPY(ADR(Get.Mobile.NetworkOperator),  ADR(arw_DataBuffer[22]), 32);
		
		get.Device.Temperature	:= 	UDINT_TO_REAL ( SHL(	WORD_TO_UDINT(	arw_DataBuffer[4]),16)	+	arw_DataBuffer[5] )/10;

		ui_MBRetryCount := 0;
		sfctip := TRUE;
	ELSE
		ui_MBRetryCount := ui_MBRetryCount + 1;
		sfctip := TRUE;
	END_IF
END_IF
END_ACTION

ACTION aReadGPSData:


MBRead(
	sIPAddr := stRouterparams.IP_TELTONIKA,
	nTCPPort := stRouterparams.MBPort_TELTONIKA,
	nUnitID := 1,
	nMBAddr := 143,
	nQuantity := 42,//*2,
	cbLength := SIZEOF(arw_DataBuffer),
	pDestAddr := ADR(arw_DataBuffer),
	bExecute := ton_GetDataTimer.Q,
	bBusy => b_busy,
	bError => b_CommError,
	nErrId => udi_errid,
	cbRead => udi_cbread,
	tTimeout := stRouterparams.T_MBTimeout
);

ftrig_TransmissionDone(clk := b_busy);

IF ftrig_TransmissionDone.q THEN
	IF NOT b_CommError THEN
		
		realconverter.Registers[2] := arw_DataBuffer[0];
		realconverter.Registers[1] := arw_DataBuffer[1];
		Get.GPS.Latitude  := realconverter.realvalue;
 
		realconverter.Registers[2] := arw_DataBuffer[2];
		realconverter.Registers[1] := arw_DataBuffer[3];
		Get.GPS.Longitude  := realconverter.realvalue;
		
		FOR ui_ForCounter := 4 TO 35 DO
			arw_DataBuffer[ui_ForCounter] := be16_TO_HOST(arw_DataBuffer[ui_ForCounter]);
		END_FOR
				
		MEMCPY(ADR(Get.GPS.FixTime),  ADR(arw_DataBuffer[4]), 32);			//GPS fixtime (text, unix timetamp * 1000)
		
		MEMCPY(ADR(Get.GPS.DateTime), ADR(arw_DataBuffer[20]), 32);			//GPS DateTime (text, YYYY-MM-DD HH:MM:SS)
		
		realconverter.Registers[2] := arw_DataBuffer[36];					//GPS speed
		realconverter.Registers[1] := arw_DataBuffer[37];
		Get.GPS.Speed  := realconverter.realvalue;
		
	
		MEMCPY(ADR(Get.GPS.SatCount)+2, ADR(arw_DataBuffer[38]), 2);			//GPS sattelite count
		MEMCPY(ADR(Get.GPS.SatCount), ADR(arw_DataBuffer[39]), 2);			//GPS sattelite count
		
		realconverter.Registers[2] := arw_DataBuffer[40];
		realconverter.Registers[1] := arw_DataBuffer[41];
		Get.GPS.Accuracy  := realconverter.realvalue;						//GPS accuracy
		
			
		ui_MBRetryCount := 0;
		sfctip := TRUE;
	ELSE
		ui_MBRetryCount := ui_MBRetryCount + 1;
		sfctip := TRUE;
	END_IF
END_IF
END_ACTION

ACTION aReadSerial:
MBRead(
	sIPAddr := stRouterparams.IP_TELTONIKA,
	nTCPPort := stRouterparams.MBPort_TELTONIKA,
	nUnitID := 1,
	nMBAddr := 39,
	nQuantity := 16,//*2,
	cbLength := SIZEOF(arw_DataBuffer),
	pDestAddr := ADR(arw_DataBuffer),
	bExecute := ton_GetDataTimer.Q,
	bBusy => b_busy,
	bError => b_CommError,
	nErrId => udi_errid,
	cbRead => udi_cbread,
	tTimeout := stRouterparams.T_MBTimeout
);

ftrig_TransmissionDone(clk := b_busy);

IF ftrig_TransmissionDone.q THEN
	IF NOT b_CommError THEN
		FOR ui_ForCounter := 0 TO 16 DO
			arw_DataBuffer[ui_ForCounter] := be16_TO_HOST(arw_DataBuffer[ui_ForCounter]);
		END_FOR
		
		//MEMCPY(ADR(Get.Mobile.NetworkOperator),  ADR(arw_DataBuffer[0]), 32);
		MEMCPY(ADR(Get.Device.RouterSerial),  ADR(arw_DataBuffer[0]), 32);
		
		ui_MBRetryCount := 0;
		sfctip := TRUE;
	ELSE
		ui_MBRetryCount := ui_MBRetryCount + 1;
		sfctip := TRUE;
	END_IF
END_IF
END_ACTION

ACTION aSendSMS:

IF get.e_SMSStatus = eSMSStatus.SendingMessage THEN
	MBSingleWrite(
		sIPAddr := stRouterparams.IP_TELTONIKA,
		nTCPPort := stRouterparams.MBPort_TELTONIKA,
		nUnitID := 1,
		nMBAddr := 396,
		nValue	:=	1,
		bExecute := ton_GetDataTimer.Q,
		bBusy => b_busy,
		bError => b_CommError,
		nErrId => udi_errid,
		tTimeout := stRouterparams.T_MBTimeout
	);
	
	ftrig_TransmissionDone(clk := b_busy);
	
	IF ftrig_TransmissionDone.q THEN
		IF NOT b_CommError THEN
			get.e_SMSStatus := eSMSSTatus.idle;
			//memcpy(ADR(get.Mobile.st_LatestSMSReceiver), ADR(ar_SMSData[0]), 20);		
			//memcpy(ADR(get.Mobile.st_LatestSMSReceiver), ADR(ar_SMSData[10]), 80);		
			ui_SMSRetryCounter := 0;
			ui_MBRetryCount := 0;
			sfctip := TRUE;
		ELSE
			ui_MBRetryCount := ui_MBRetryCount + 1;
			ui_SMSRetryCounter := ui_SMSRetryCounter + 1;
			IF ui_SMSRetryCounter > 0 THEN
				get.Events.b_SMSNotSendError := TRUE;
				get.e_SMSStatus := eSMSStatus.error;
				sfctip := TRUE;
			END_IF
		END_IF
	END_IF
ELSE
	SFCtip := NOT SFCTip;
END_IF
END_ACTION

ACTION aWriteSMSData:

MBWrite(
	sIPAddr := stRouterparams.IP_TELTONIKA,
	nTCPPort := stRouterparams.MBPort_TELTONIKA,
	nUnitID := 1,
	nMBAddr := 397,
	nQuantity := 90,
	cbLength := SIZEOF(ar_SMSData),
	pSrcAddr	:=	ADR(ar_SMSData),
	bExecute := ton_GetDataTimer.Q,
	bBusy => b_busy,
	bError => b_CommError,
	nErrId => udi_errid,
	tTimeout := stRouterparams.T_MBTimeout
);

ftrig_TransmissionDone(clk := b_busy);

IF ftrig_TransmissionDone.q THEN
	IF NOT b_CommError THEN
		get.e_SMSStatus := eSMSStatus.SendingMessage;
		ui_SMSRetryCounter := 0;
		ui_MBRetryCount := 0;
		sfctip := TRUE;
	ELSE
		ui_SMSRetryCounter := ui_SMSRetryCounter +1;
		ui_MBRetryCount := ui_MBRetryCount + 1;
		IF ui_SMSRetryCounter > 3 THEN
			get.Events.b_SMSNotSendError := TRUE;
			get.e_SMSStatus := eSMSStatus.error;
			sfctip := TRUE;
		END_IF
	END_IF
END_IF
END_ACTION

METHOD CreateMessage : BOOL
VAR_INPUT
//	TelNumber	:	ULINT;
	s_Message		:	STRING(80);
END_VAR

VAR
	s_InternalMessage 	: 	STRING(160);
	s_LAT				:	STRING(8);
	s_LONG				:	STRING(9);
	ui_counter			:	UINT;
END_VAR

memcpy(ADR(ar_SMSData[0]), ADR(get.Mobile.s_EmergencySMSNumber), 20);

s_LAT := REAL_TO_STRING(get.GPS.Latitude);
s_LONG := REAL_TO_STRING(get.GPS.Longitude);

s_InternalMessage := 'ePU10 LFP Battery System Alarm';
s_InternalMessage := concat(s_InternalMessage, '$n');
s_InternalMessage := concat(s_InternalMessage, 'ID: ');
s_InternalMessage := concat(s_InternalMessage, get.mobile.s_EmergencySMSDevName);
s_InternalMessage := concat(s_InternalMessage, '$n');
s_InternalMessage := concat(s_InternalMessage, 'LAT: ');
s_InternalMessage := concat(s_InternalMessage, s_LAT);
s_InternalMessage := concat(s_InternalMessage, '$n');
s_InternalMessage := concat(s_InternalMessage, 'LON: ');
s_InternalMessage := concat(s_InternalMessage, s_LONG);
s_InternalMessage := concat(s_InternalMessage, '$n');
s_InternalMessage := concat(s_InternalMessage,s_Message);

memcpy(ADR(ar_SMSData[10]), ADR(s_InternalMessage[0]), 160);

FOR ui_counter := 0 TO 89 DO
	ar_SMSData[ui_counter] := host_to_be16(ar_SMSData[ui_counter]);
END_FOR

CreateMessage := TRUE;
END_METHOD

METHOD EMStop : BOOL
VAR_INPUT
END_VAR

//nothing to do here
EMSTOP := TRUE;
END_METHOD

METHOD GetDiagnostics : BOOL
VAR_INPUT
END_VAR
END_METHOD

ACTION ReadDataSFC:
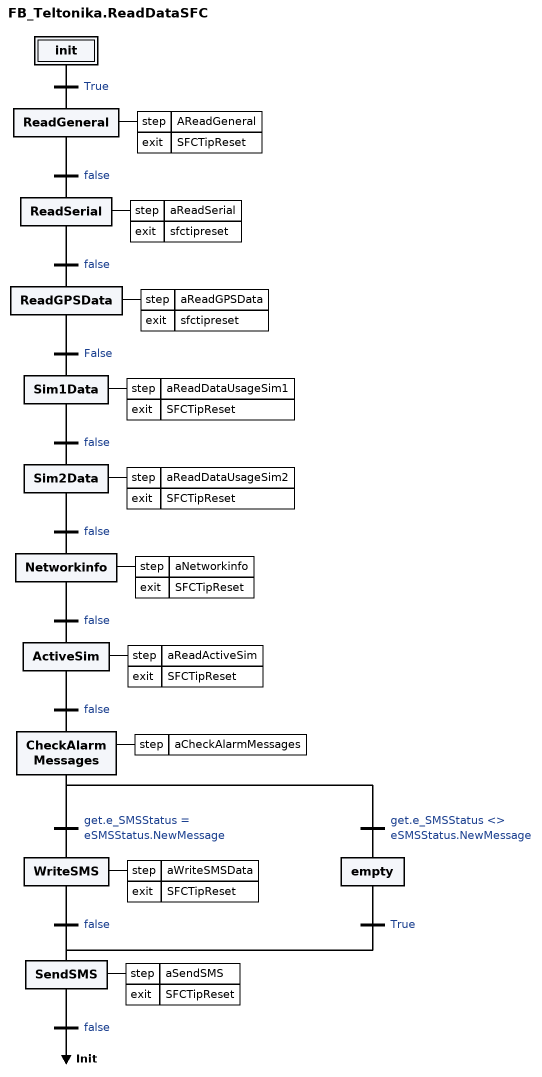
INITIAL_STEP init:
END_STEP
TRANSITION FROM init TO ReadGeneral
    := True;
END_TRANSITION
STEP ReadGeneral:
    AReadGeneral(N);  // step action
    SFCTipReset(P0);  // exit action
END_STEP
TRANSITION FROM ReadGeneral TO ReadSerial
    := false;
END_TRANSITION
STEP ReadSerial:
    aReadSerial(N);  // step action
    sfctipreset(P0);  // exit action
END_STEP
TRANSITION FROM ReadSerial TO ReadGPSData
    := false;
END_TRANSITION
STEP ReadGPSData:
    aReadGPSData(N);  // step action
    sfctipreset(P0);  // exit action
END_STEP
TRANSITION FROM ReadGPSData TO Sim1Data
    := False;
END_TRANSITION
STEP Sim1Data:
    aReadDataUsageSim1(N);  // step action
    SFCTipReset(P0);  // exit action
END_STEP
TRANSITION FROM Sim1Data TO Sim2Data
    := false;
END_TRANSITION
STEP Sim2Data:
    aReadDataUsageSim2(N);  // step action
    SFCTipReset(P0);  // exit action
END_STEP
TRANSITION FROM Sim2Data TO Networkinfo
    := false;
END_TRANSITION
STEP Networkinfo:
    aNetworkinfo(N);  // step action
    SFCTipReset(P0);  // exit action
END_STEP
TRANSITION FROM Networkinfo TO ActiveSim
    := false;
END_TRANSITION
STEP ActiveSim:
    aReadActiveSim(N);  // step action
    SFCTipReset(P0);  // exit action
END_STEP
TRANSITION FROM ActiveSim TO CheckAlarmMessages
    := false;
END_TRANSITION
STEP CheckAlarmMessages:
    aCheckAlarmMessages(N);  // step action
END_STEP
TRANSITION FROM CheckAlarmMessages TO WriteSMS
    := get.e_SMSStatus = eSMSStatus.NewMessage;
END_TRANSITION
STEP WriteSMS:
    aWriteSMSData(N);  // step action
    SFCTipReset(P0);  // exit action
END_STEP
TRANSITION FROM WriteSMS TO SendSMS
    := false;
END_TRANSITION
TRANSITION FROM CheckAlarmMessages TO empty
    := get.e_SMSStatus <> eSMSStatus.NewMessage;
END_TRANSITION
STEP empty:
END_STEP
TRANSITION FROM empty TO SendSMS
    := True;
END_TRANSITION
STEP SendSMS:
    aSendSMS(N);  // step action
    SFCTipReset(P0);  // exit action
END_STEP
TRANSITION FROM SendSMS TO Init
    := false;
END_TRANSITION
// branch label Branch0_ReadDataSFC
END_ACTION

METHOD Reset : BOOL
VAR_INPUT
END_VAR

get.Events.b_MBCommError := FALSE;
get.Events.b_MBCommError := FALSE;
get.Events.b_SMSNotSendError := FALSE;
get.e_SMSStatus := eSMSStatus.Idle;

Reset := TRUE;
END_METHOD

METHOD SetDevName : BOOL
VAR_INPUT
	s_DevName	:	String(12);
END_VAR
IF s_DevName = '' THEN
	get.Mobile.s_EmergencySMSDevName := 'serial'; //<-- stParams.serial number
ELSE
	get.Mobile.s_EmergencySMSDevName :=	s_DevName;
END_IF

SetDevName := True;
END_METHOD

METHOD SetSMSNumber : BOOL
VAR_INPUT
	s_SMSNumber	:	STRING(20);
END_VAR
VAR 
	for_counter	:	UINT :=0;
	InternalString	:	STRING(20);
	intermediateValue	:	UINT;
	
	temp	:	string(10);
END_VAR

SetSMSNumber := TRUE;

//check minimum length
IF INT_TO_UINT(len(s_SMSNumber)) < stRouterParams.MinimumPhoneNumberLength THEN
	SetSMSNumber := FALSE;
ELSE
	InternalString := s_SMSNumber;
	
	//replace leading + with 00
	IF left(InternalString,1) = '+' THEN
		InternalString := Replace(InternalString, '00', 1, 1);
	END_IF
	
	//check for non_numeric characters
	FOR for_counter := 1 TO INT_TO_UINT(len(InternalString)) DO
		intermediateValue := f_toASC(mid(InternalString, 1, UINT_TO_INT(for_counter)));
		IF (intermediateValue < 48 OR intermediateValue > 57) THEN
			SetSMSNumber := FALSE;
		END_IF
	END_FOR
END_IF

//only if all checks succeed, the number is written to the struct.
IF SetSMSNumber THEN
	get.Mobile.s_EmergencySMSNumber := InternalString;
END_IF
END_METHOD

ACTION SFCTipReset:
SFCTip := FALSE;
END_ACTION

END_FUNCTION_BLOCK

// ---- POUs/Objects/LedstripController/UpdateSFC.TcPOU
FUNCTION_BLOCK UpdateSFC
VAR
	stSystemState	:	ST_Ledstrip_IOvars;
	r_SOC			:	REAL;
	r_Powerload		:	REAL;
	AnimationIndex: UINT;
END_VAR


VAR
	B_Update			: 	BOOL;
	ton_UpdateTimer		:	TON;
	ton_SOCUpdateTimer		:	TON;
	ton_AnimationUpdateTimer		:	TON;
	ftrig_Execute		:	f_trig;//TP := (PT := T#50MS);
	
	u_CurrentLEDColor		:	u_LedColor;
	
	FBRand	:	DRAND();
	seed	:	INT;
	
	Animation		:   UINT := 0;

	ChargeState		:	UINT;	//0=idle, 1=charging, 2=discharging
	
	st_Control		AT %Q*	:	stLedControl;
	st_Status		AT %I* :	stLedStatus;
	fTrig_CommandReady		:	f_trig;
	
	Param_AnimationLength			:	USINT		:=	5;
	Param_NrOfLeds					:	USINT 		:=	120;
	Param_UpdateInterval			:	TIME		:=	T#100MS;
	Param_AnimationUpdateInterval	:	TIME		:=	T#500MS;
	Param_SOCUpdateInterval			:	TIME		:=	T#1000MS;
	Param_EnablePowerLevel			:	BOOL		:=	TRUE;	
	params_CurrentTriggerlevel		:	INT			:=	10;
	by_LedIntensity					:	BYTE		:= 	127;
	
	UI_SOCLedIndex					: 	UINT;
	UI_PowerLevelIndex				:	UINT;
END_VAR

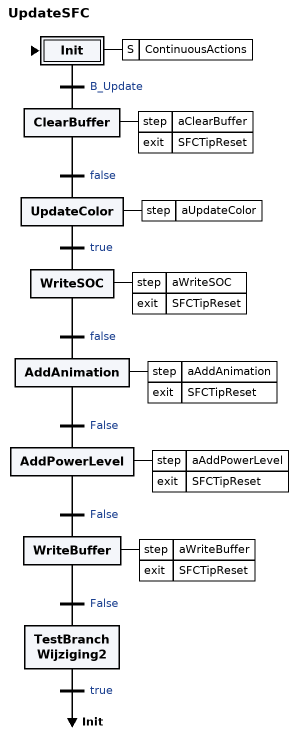
INITIAL_STEP Init:
    ContinuousActions(S);
END_STEP
TRANSITION FROM Init TO ClearBuffer
    := B_Update;
END_TRANSITION
STEP ClearBuffer:
    aClearBuffer(N);  // step action
    SFCTipReset(P0);  // exit action
END_STEP
TRANSITION FROM ClearBuffer TO UpdateColor
    := false;
END_TRANSITION
STEP UpdateColor:
    aUpdateColor(N);  // step action
END_STEP
TRANSITION FROM UpdateColor TO WriteSOC
    := true;
END_TRANSITION
STEP WriteSOC:
    aWriteSOC(N);  // step action
    SFCTipReset(P0);  // exit action
END_STEP
TRANSITION FROM WriteSOC TO AddAnimation
    := false;
END_TRANSITION
STEP AddAnimation:
    aAddAnimation(N);  // step action
    SFCTipReset(P0);  // exit action
END_STEP
TRANSITION FROM AddAnimation TO AddPowerLevel
    := False;
END_TRANSITION
STEP AddPowerLevel:
    aAddPowerLevel(N);  // step action
    SFCTipReset(P0);  // exit action
END_STEP
TRANSITION FROM AddPowerLevel TO WriteBuffer
    := False;
END_TRANSITION
STEP WriteBuffer:
    aWriteBuffer(N);  // step action
    SFCTipReset(P0);  // exit action
END_STEP
TRANSITION FROM WriteBuffer TO TestBranchWijziging2
    := False;
END_TRANSITION
STEP TestBranchWijziging2:
END_STEP
TRANSITION FROM TestBranchWijziging2 TO Init
    := true;
END_TRANSITION

ACTION aAddAnimation:

IF ChargeState = 0 THEN
	st_Control.b_Execute :=	FALSE;
	SFCTip := NOT SFCTip;
ELSE
	st_Control.by_Command := 1;
	st_Control.w_Index	:=	AnimationIndex;
	st_Control.w_Length	:=	1;
	st_Control.dw_Color :=  u_CurrentLEDColor.dw_LedColor;
	st_Control.b_Execute 	:=	NOT st_Control.b_Execute;
	
	IF ftrig_CommandReady.Q THEN
		st_Control.b_Execute :=	FALSE;
		SFCTip := TRUE;
	END_IF
END_IF
END_ACTION

ACTION aAddPowerLevel:
UI_PowerLevelIndex := LIMIT(1, REAL_TO_WORD((USINT_TO_REAL(Param_NrOfLeds)/100*r_Powerload)), USINT_TO_WORD(Param_NrOfLeds));

st_Control.by_Command := 1;
st_Control.w_Index	:=	UI_PowerLevelIndex;
st_Control.w_Length	:=	1;//UI_SOCLedIndex;
st_Control.dw_Color := 16#007F0000;
st_Control.b_Execute 	:=	NOT st_Control.b_Execute;

IF ftrig_CommandReady.Q THEN
	st_Control.b_Execute :=	FALSE;
	SFCTip := TRUE;
END_IF
END_ACTION

ACTION aClearBuffer:
b_update := FALSE;

st_Control.by_Command 	:= 	2;
st_Control.b_Execute 	:=	NOT st_Control.b_Execute;

IF ftrig_CommandReady.Q THEN
	st_Control.b_Execute :=	FALSE;
	SFCTip := TRUE;
END_IF

//testbrancheWijziging1
END_ACTION

ACTION aUpdateColor:

IF stSystemState.b_Error THEN
	u_CurrentLEDColor.st_LedColor.by_Red := by_LedIntensity;
	u_CurrentLEDColor.st_LedColor.by_Green := 0;
	u_CurrentLEDColor.st_LedColor.by_Blue := 0;
	u_CurrentLEDColor.st_LedColor.by_White := 0;
ELSIF stSystemState.b_warning THEN
	u_CurrentLEDColor.st_LedColor.by_Red := by_LedIntensity/2;
	u_CurrentLEDColor.st_LedColor.by_Green := by_LedIntensity/2;
	u_CurrentLEDColor.st_LedColor.by_Blue := 0;
	u_CurrentLEDColor.st_LedColor.by_White := 0;
ELSIF stSystemState.b_attention THEN
	u_CurrentLEDColor.st_LedColor.by_Red := 0;
	u_CurrentLEDColor.st_LedColor.by_Green := 0;
	u_CurrentLEDColor.st_LedColor.by_Blue := 0;
	u_CurrentLEDColor.st_LedColor.by_White := by_LedIntensity/2;	
ELSIF stSystemState.b_normal THEN
	u_CurrentLEDColor.st_LedColor.by_Red := 0;
	u_CurrentLEDColor.st_LedColor.by_Green := by_LedIntensity;
	u_CurrentLEDColor.st_LedColor.by_Blue := 0;
	u_CurrentLEDColor.st_LedColor.by_White := 0;
ELSE
	u_CurrentLEDColor.st_LedColor.by_Red := 0;
	u_CurrentLEDColor.st_LedColor.by_Green := 0;
	u_CurrentLEDColor.st_LedColor.by_Blue := by_LedIntensity;
	u_CurrentLEDColor.st_LedColor.by_White := 0;
END_IF
END_ACTION

ACTION aWriteBuffer:
st_Control.b_Update		:= TRUE;
st_Control.b_send		:= TRUE;
st_Control.b_Execute 	:=	NOT st_Control.b_Execute;

IF ftrig_CommandReady.Q THEN
	st_Control.b_Execute :=	FALSE;
	st_Control.b_Update		:= FALSE;
	st_Control.b_send		:= FALSE;
	SFCTip := TRUE;
END_IF
END_ACTION

ACTION aWriteSOC:
UI_SOCLedIndex := LIMIT(1, REAL_TO_WORD((USINT_TO_REAL(Param_NrOfLeds)/100*r_SOC)), USINT_TO_WORD(Param_NrOfLeds));

st_Control.by_Command := 1;
st_Control.w_Index	:=	0;
st_Control.w_Length	:=	UI_SOCLedIndex;
st_Control.dw_Color := u_CurrentLEDColor.dw_LedColor;
st_Control.b_Execute 	:=	NOT st_Control.b_Execute;

IF ftrig_CommandReady.Q THEN
	st_Control.b_Execute :=	FALSE;
	SFCTip := TRUE;
END_IF
END_ACTION

ACTION ContinuousActions:

ton_UpdateTimer(in := NOT ton_UpdateTimer.Q, PT := Param_UpdateInterval);

IF ton_UpdateTimer.Q THEN
	B_Update := TRUE;
END_IF

fTrig_CommandReady(Clk := st_Control.b_Execute);//st_Status.b_busy);

IF stSystemState.r_DCCurrent > params_CurrentTriggerlevel THEN
	ChargeState := 2;
ELSIF 	stSystemState.r_DCCurrent < (-params_CurrentTriggerlevel) THEN
	ChargeState := 1;
ELSE
	ChargeState := 0;
END_IF



ton_AnimationUpdateTimer(in := NOT ton_AnimationUpdateTimer.Q, PT := Param_AnimationUpdateInterval);
IF ton_AnimationUpdateTimer.q THEN
	CASE ChargeState OF
		0:
			AnimationIndex := UI_SOCLedIndex;// + Animation

			
		1: 
			IF AnimationIndex <= UI_SOCLedIndex THEN
				AnimationIndex := UI_SOCLedIndex + Param_AnimationLength-1;
				//Animation := Param_AnimationLength-1;
			ELSE
				AnimationIndex := AnimationIndex-1;
			END_IF
			
		2: 
			IF AnimationIndex >= UI_SOCLedIndex + Param_AnimationLength-1 THEN
				AnimationIndex := UI_SOCLedIndex;
			ELSE
				AnimationIndex := AnimationIndex+1;
			END_IF
	END_CASE
END_IF

FBRand(Seed := Seed);
ton_SOCUpdateTimer(in := NOT ton_SOCUpdateTimer.Q, PT := Param_SOCUpdateInterval);

IF ton_SOCUpdateTimer.Q THEN
	IF r_SOC < 0 THEN
		stSystemState.r_DCCurrent := -stSystemState.r_DCCurrent;
		r_SOC := 0;
	ELSIF r_SOC > 100 THEN
		stSystemState.r_DCCurrent := -stSystemState.r_DCCurrent;
		r_SOC := 100;
	ELSE
		r_SOC := r_SOC - (stSystemState.r_DCCurrent / (63 * 36));
	END_IF


	IF stSystemState.r_DCCurrent > 0 THEN
		stSystemState.r_DCCurrent := LIMIT(20, stSystemState.r_DCCurrent + ((FBRand.Num-0.5)*100), 630);
	ELSIF stSystemState.r_DCCurrent < 0 THEN
		stSystemState.r_DCCurrent := LIMIT(-630, stSystemState.r_DCCurrent + ((FBRand.Num-0.5)*100), -20);
	END_IF

	r_Powerload := ABS(stSystemState.r_DCCurrent/630)*100; 
	
END_IF
END_ACTION

ACTION SFCTipReset:
SFCTip := FALSE;
st_Control.b_Execute 	:= FALSE;
st_Control.b_Update		:= FALSE;
st_Control.b_send		:= FALSE;
END_ACTION

END_FUNCTION_BLOCK

// ---- POUs/ErrorHandling/ErrorHandling.TcPOU
PROGRAM INTERNAL ErrorHandling
VAR_INPUT
	e_access					: eErrAckAccess;
	AddError					: ARRAY [0..i_maxevents] OF FB_addErrorST;
END_VAR

VAR	
	//Errorhandling
	w_ErrorIndex				: WORD;
	b_ClearEvents				: BOOL;	
	b_ResetError				: BOOL;
	(*ENUM*)
	
	//autoclear pulse
	ton_AutoResetClear 						: TON :=(PT:= T#1S);
	//Refresh Timer
	ton_RefreshTimer						: TON := (PT:= T#10S);
	b_refreshErrors							: BOOL;
END_VAR

VAR_OUTPUT
	{ attribute 'TcHmiSymbol.ShowRecursively' }
	a_ActiveEvents						: ARRAY [0..i_maxevents	] OF ST_ErrorStruct;
	w_errorword							: WORD;
	b_errorActive						: BOOL;
END_VAR

VAR CONSTANT
	i_maxevents							: INT := 200;
END_VAR

//Reset variables
w_ErrorIndex 					:= 0;

//RealtimeClock
//SystemClock();

//Autoreset signal
ton_AutoResetClear(IN:= NOT(ton_AutoResetClear.Q));

//EventLogger
//fbAlarm(evtEntry := TC_Events.myWarningEventClass.Warning, bEvt:=b_event, bClear := b_Clear);

//Refresh signal
ton_RefreshTimer(IN:= NOT(ton_RefreshTimer.Q));
b_RefreshErrors := ton_RefreshTimer.Q OR GVL.b_InitCycle;
IF b_RefreshErrors THEN
	GVL.b_WarningActive				:= FALSE;
	GVL.b_NormalShutdownActive		:= FALSE;
	GVL.b_QuickshutdownActive		:= FALSE;
	GVL.b_EmergencyShutdownActive	:= FALSE;	

